(* IEC 61131-3 sources: elnaProjects/ElpcLogic/PomarKc7Changed/build_USO_ecl/_ (part 4) *)

  	IF StrSw.reliability THEN
  		IF _statOn AND NOT _statOff 		THEN 	StrSw.onStatus := _statusDualInput.STATUS_ON;
  		ELSIF _statOff AND NOT _statOn 	THEN 	StrSw.onStatus := _statusDualInput.Status_OFF;
  		ELSIF NOT _statOn AND NOT _statOff 	THEN 	StrSw.onStatus := _statusDualInput.STATUS_TRANSITIONAL;
  		ELSE					StrSw.onStatus := _statusDualInput.STATUS_ERROR;
                      END_IF;

  	ELSE
  		StrSw.onStatus := _statusDualInput.STATUS_NOTDEFINED;

  	END_IF;
  ELSE
  	CASE BYTE_TO_INT(lastCmd) OF
  		(*baseCmdOn*) 1: StrSw.onStatus  := _statusDualInput.STATUS_ON;
  		(*baseCmdOff*) 2: StrSw.onStatus  := _statusDualInput.STATUS_OFF;

  	ELSE
  		 StrSw.onStatus := _statusDualInput.STATUS_NOTDEFINED;

  	END_CASE;
  END_IF;

  StrSw.Accident := inAccident.value AND inAccident.reliability;
  StrSw.Ns := inNs.value AND inNs.reliability;
  StrSw.Local := inLocal.value AND inLocal.reliability;
  StrSw.Distance := inDistance.value AND inDistance.reliability;
  StrSw.OpcCommandsDisabled := StrSw.inOpcCommandsDisabled;

  StrSw.Blocked:=StrSw.Accident OR StrSw.Local OR StrSw.breakCmdOn OR StrSw.breakCmdOff OR StrSw.inBlocked;

  StrSw.Rezervny:=NOT StrSw.Osnovnoy;

  (* ---- Формирование признака сдвига ---- *)

  getSdvig := FALSE;
  IF (StrSw.ISVALIDREF_cmdOn OR StrSw.ISVALIDREF_cmdOff) AND NOT StrSw.Local THEN
  	IF NOT (StrSw.CmdOn OR StrSw.CmdOff) THEN
                       IF (lastOnStatus <> StrSw.onStatus AND
  		(StrSw.onStatus <> _statusDualInput.STATUS_NOTDEFINED AND
                       StrSw.onStatus <> _statusDualInput.STATUS_ERROR)     AND
  		(lastOnStatus <> _statusDualInput.STATUS_NOTDEFINED   AND
                       lastOnStatus <> _statusDualInput.STATUS_ERROR))
                      THEN
  			getSdvig   := TRUE;
  		END_IF;
  	END_IF;
  END_IF;

  IF getSdvig THEN StrSw.sdvig:= TRUE; END_IF;

  sdvigReset(IN:=StrSw.sdvig, PT:=T#15S);

  IF sdvigReset.Q THEN StrSw.sdvig:=FALSE; END_IF;

  lastOnStatus := StrSw.onStatus;

  (* ---- Распаковка команды ---- *)
  _sunpackerCommand(command := StrSw.inCommand);
  	cmd := _sunpackerCommand.cmd;
  	source := _sunpackerCommand.source;

  (* ---- Обработка команды ---- *)
  IF cmd <> 0 AND lastCmd <> cmd and (((NOT StrSw.opcCommandsDisabled) AND source > 0) OR source = 0) then
  	CASE BYTE_TO_INT(cmd) OF
  	(*cmd_on*) 1 :
  			IF  StrSw.ISVALIDREF_cmdOn THEN StrSw.CmdOn := TRUE;
  				IF StrSw.ISVALIDREF_cmdOff THEN StrSw.CmdOff := FALSE; END_IF;
  			ELSIF  StrSw.ISVALIDREF_cmdOff THEN StrSw.CmdOff := FALSE;  END_IF;
  			errorCMDTimer(IN := false);
  			_commandErrorTimer := true;
  			StrSw.lastCmdIsOn := true;
  	(*cmd_off*) 2 :
  			IF StrSw.ISVALIDREF_cmdOff THEN StrSw.CmdOff := TRUE;
  				IF StrSw.ISVALIDREF_cmdOn THEN StrSw.CmdOn := FALSE; END_IF;
  			ELSIF StrSw.ISVALIDREF_cmdOn THEN StrSw.CmdOn := FALSE; END_IF;
  			errorCMDTimer(IN := false);

  			_commandErrorTimer := true;
  			StrSw.lastCmdIsOn := false;
  	(*cmd_reset*) 3 :    IF StrSw.ISVALIDREF_statOn OR StrSw.ISVALIDREF_statOff THEN
  			StrSw.CmdOn := FALSE;
  			StrSw.CmdOff := FALSE;
                                lastCmd := 0;
  			_commandErrorTimer := false;
  			StrSw.lastCmdIsOn := false;
                                 END_IF;
  	END_CASE;
  	source_for_Status := source;
  	cmd_for_Status := cmd;
  	command_error_for_Status := 0;
  END_IF;

  lastCmd := cmd;
  errorCMDTimer(In := _commandErrorTimer, PT :=T#10s);

  (* ---- алгоритм  для команды ВКЛючить ---- *)
  IF (StrSw.onStatus = _statusDualInput.STATUS_ON) and StrSw.lastCmdIsOn then
  	IF StrSw.ISVALIDREF_cmdOn AND StrSw.ISVALIDREF_cmdOff then  StrSw.cmdOn := false; END_IF;

  	 errorCMDTimer(In := false);
  	 _commandErrorTimer := false;
  	 cmd_for_Status := 0;
  	 source_for_Status := 0;
  END_IF;

  (* ---- off ---- *)
  IF (StrSw.onStatus = _statusDualInput.STATUS_OFF) and (NOT StrSw.lastCmdIsOn) then
  	IF StrSw.ISVALIDREF_cmdOn AND StrSw.ISVALIDREF_cmdOff then  StrSw.cmdOff := false; END_IF;

  	 errorCMDTimer(In := false);
  	 _commandErrorTimer := false;
  	 cmd_for_Status := 0;
  	 source_for_Status := 0;
  END_IF;

  (* ---- ошибка исполнения команды ---- *)
  if errorCMDTimer.Q and (cmd_for_Status <> 0) then
  	command_error_for_Status :=  cmd_for_Status;
  	_commandErrorTimer := false;
  	StrSw.CmdOn := false;
  	StrSw.CmdOff := false;
  	lastCmd := 0;
  end_if;

  (* ---- сброс ошибки команды ---- *)
  StrSw.CommandFault := command_error_for_Status <> 0;
  _errorReset(IN := command_error_for_Status <> 0, PT := T#5S);
  IF _errorReset.Q THEN
  	cmd_for_Status := 0;
  	source_for_Status := 0;
  	command_error_for_Status := 0;
  END_IF;

  outputsSets(in := (StrSw.ISVALIDREF_cmdOn and StrSw.cmdOn ) OR (StrSw.ISVALIDREF_cmdOff and StrSw.cmdOff), PT := T#2S);
  	IF NOT outputsSets.Q THEN
  		StrSw.BreakCmdOn := inBreakCmdOn._inversed AND inBreakCmdOn.reliability AND StrSw.ISVALIDREF_inBreakCmdOn;
  		StrSw.BreakCmdOff := inBreakCmdOff._inversed AND inBreakCmdOff.reliability AND StrSw.ISVALIDREF_inBreakCmdOff;
  	END_IF;

  cmdOn := StrSw.cmdOn;
  cmdOff:= StrSw.cmdOff;

  (* ---- формирование зашифрованного статуса для АРМа ---- *)
  StrSw.status := shl(BYTE_TO_DWORD(source_for_Status), 29)
  		OR shl(BYTE_TO_DWORD(cmd_for_Status), 26)
  		OR shl(BYTE_TO_DWORD(command_error_for_Status), 23)
  		OR shl(bool_to_DWORD(StrSw.sdvig), 22)
  		OR shl(bool_to_DWORD(StrSw.OpcCommandsDisabled), 21)
                      OR shl(bool_to_DWORD(StrSw.lastCmdIsOn), 14)
                      OR shl(BOOL_TO_DWORD(StrSw.BreakCmdOff), 13)
  		OR shl(BOOL_TO_DWORD(StrSw.BreakCmdOn), 12)
  		OR shl(BOOL_TO_DWORD(StrSw.Distance), 6)
  		OR shl(BOOL_TO_DWORD(StrSw.Local), 5)
  		OR shl(BOOL_TO_DWORD(StrSw.Ns), 4)
                  	OR shl(BOOL_TO_DWORD(StrSw.Accident ),3)
  		OR BYTE_TO_DWORD(StrSw.onStatus);
END_FUNCTION_BLOCK

FUNCTION_BLOCK fb_Switch
  VAR_INPUT
    statOn : BOOL;
    statOff : BOOL;
    statOn_reliability : BOOL;
    statOff_reliability : BOOL;
  END_VAR
  VAR_IN_OUT
    StrSw : struct_Switch;
  END_VAR
  VAR_INPUT
    inNs : TYPE_ReliableBit;
    inAccident : TYPE_ReliableBit;
    inAuto : TYPE_ReliableBit;
    inManual : TYPE_ReliableBit;
    inLocal : TYPE_ReliableBit;
    inDistance : TYPE_ReliableBit;
    inErrorPowerOff : TYPE_ReliableBit;
    inErrorBlock : TYPE_ReliableBit;
    inBreakCmdOn : TYPE_ReliableBit;
    inBreakCmdOff : TYPE_ReliableBit;
  END_VAR
  VAR
    onInit : BOOL      := FALSE;
    _statOn : BOOL;
    _statOff : BOOL;
    lastOnStatus : BYTE;
    cmd : BYTE;
    source : BYTE;
    lastCmd : BYTE;
    source_for_Status : BYTE;
    cmd_for_Status : BYTE;
    command_error_for_Status : BYTE;
    _sunpackerCommand : fb_sunpackerCommand;
    _statusDualInput : TYPE_statusDualInput;
    _commandDualInput : TYPE_commandDualInput;
    _commandErrorTimer : BOOL;
    resetErrorTimer : BOOL;
    getSdvig : BOOL;
    _changWithoutCommand : BOOL;
    errorCMDTimer : TON;
    sdvigReset : TON;
    _errorReset : TON;
    outputsSets : TOF;
  END_VAR
  VAR_IN_OUT
    cmdOn : BOOL;
    cmdOff : BOOL;
  END_VAR

  IF NOT onInit THEN
  IF StrSw.ISVALIDREF_cmdOn XOR StrSw.ISVALIDREF_cmdOff THEN
  	IF 	StrSw.ISVALIDREF_cmdOn THEN
  		lastCmd:= 2; (*baseCmdOff*)
  	ELSE
  		lastCmd:= 1; (*baseCmdOn*)
  	END_IF;
  END_IF;
  onInit:=TRUE;
  END_IF;

  (* ---- Если управление с ВУ заблокировано, то в ИМ передаем команду из алгоритма ---- *)
  IF StrSw.inOpcCommandsDisabled THEN
  	StrSw.inCommand := StrSw.inCommand_Alg;
  ELSE (* иначе передаем команду с АРМа*)
  	StrSw.inCommand := StrSw.inCommand_ARM;
  END_IF;

  (* ---- Формирование состояния механизма ---- *)

  IF (StrSw.ISVALIDREF_statOn) OR (StrSw.ISVALIDREF_statOff) THEN
  	IF (StrSw.ISVALIDREF_statOn) AND (StrSw.ISVALIDREF_statOff) THEN
  	StrSw.reliability:= statOn_reliability AND statOff_reliability;
  		_statOn  := statOn;
  		_statOff := statOff;
  	ELSIF (StrSw.ISVALIDREF_statOn) THEN
                       StrSw.reliability:= statOn_reliability;
  		_statOn  := statOn;
  		_statOff := NOT statOn;
  	ELSIF (StrSw.ISVALIDREF_statOff) THEN
  		 StrSw.reliability:= statOff_reliability;
  		_statOn  := NOT statOff;
  		_statOff :=statOff;
  	END_IF;

  	IF StrSw.reliability THEN
  		IF _statOn AND NOT _statOff 		THEN 	StrSw.onStatus := _statusDualInput.STATUS_ON;
  		ELSIF _statOff AND NOT _statOn 	THEN 	StrSw.onStatus := _statusDualInput.Status_OFF;
  		ELSIF NOT _statOn AND NOT _statOff 	THEN 	StrSw.onStatus := _statusDualInput.STATUS_TRANSITIONAL;
  		ELSE					StrSw.onStatus := _statusDualInput.STATUS_ERROR;
                      END_IF;

  	ELSE
  		StrSw.onStatus := _statusDualInput.STATUS_NOTDEFINED;

  	END_IF;
  ELSE
  	CASE BYTE_TO_INT(lastCmd) OF
  		(*baseCmdOn*) 1: StrSw.onStatus  := _statusDualInput.STATUS_ON;
  		(*baseCmdOff*) 2: StrSw.onStatus  := _statusDualInput.STATUS_OFF;

  	ELSE
  		 StrSw.onStatus := _statusDualInput.STATUS_NOTDEFINED;

  	END_CASE;
  END_IF;

  StrSw.Accident := inAccident.value AND inAccident.reliability;
  StrSw.Ns := inNs.value AND inNs.reliability;
  StrSw.Auto := inAuto.value AND inAuto.reliability;
  StrSw.Manual := inManual.value AND inManual.reliability;
  StrSw.Local := inLocal.value AND inLocal.reliability;
  StrSw.Distance := inDistance.value AND inDistance.reliability;
  StrSw.ErrorPowerOff := inErrorPowerOff.value AND inErrorPowerOff.reliability;
  StrSw.ErrorBlock := inErrorBlock.value AND inErrorBlock.reliability;
  StrSw.OpcCommandsDisabled := StrSw.inOpcCommandsDisabled;

  (* ---- Формирование признака сдвига ---- *)
  getSdvig := FALSE;
  IF (StrSw.ISVALIDREF_cmdOn OR StrSw.ISVALIDREF_cmdOff) AND NOT StrSw.Local THEN
  	IF NOT (StrSw.CmdOn OR StrSw.CmdOff) THEN
                       IF (lastOnStatus <> StrSw.onStatus AND
  		(StrSw.onStatus <> _statusDualInput.STATUS_NOTDEFINED AND
                       StrSw.onStatus <> _statusDualInput.STATUS_ERROR)     AND
  		(lastOnStatus <> _statusDualInput.STATUS_NOTDEFINED   AND
                       lastOnStatus <> _statusDualInput.STATUS_ERROR))
                      THEN
  			getSdvig   := TRUE;
  		END_IF;
  	END_IF;
  END_IF;

  IF getSdvig THEN StrSw.sdvig:= TRUE; END_IF;

  sdvigReset(IN:=StrSw.sdvig, PT:=T#15S);

  IF sdvigReset.Q THEN StrSw.sdvig:=FALSE; END_IF;

  lastOnStatus := StrSw.onStatus;

  (* ---- Распаковка команды ---- *)
  _sunpackerCommand(command := StrSw.inCommand);
  	cmd := _sunpackerCommand.cmd;
  	source := _sunpackerCommand.source;

  (* ---- Обработка команды ---- *)
  IF cmd <> 0 AND lastCmd <> cmd and (((NOT StrSw.opcCommandsDisabled) AND source > 0) OR source = 0) then
  	CASE BYTE_TO_INT(cmd) OF
  	(*cmd_open*) 1 :
  			IF  StrSw.ISVALIDREF_cmdOn THEN StrSw.CmdOn := TRUE;
  				IF StrSw.ISVALIDREF_cmdOff THEN StrSw.CmdOff := FALSE; END_IF;
  			ELSIF  StrSw.ISVALIDREF_cmdOff THEN StrSw.CmdOff := FALSE;  END_IF;
                                lastCmd := cmd;
  			errorCMDTimer(IN := false);
  			_commandErrorTimer := true;
  			StrSw.lastCmdIsOn := true;
  	(*cmd_close*) 2 :
  			IF StrSw.ISVALIDREF_cmdOff THEN StrSw.CmdOff := TRUE;
  				IF StrSw.ISVALIDREF_cmdOn THEN StrSw.CmdOn := FALSE; END_IF;
  			ELSIF StrSw.ISVALIDREF_cmdOn THEN StrSw.CmdOn := FALSE; END_IF;
                                lastCmd := cmd;
  			errorCMDTimer(IN := false);
  			_commandErrorTimer := true;
  			StrSw.lastCmdIsOn := false;
  	(*cmd_reset*) 3 :    IF StrSw.ISVALIDREF_statOn OR StrSw.ISVALIDREF_statOff THEN
  			StrSw.CmdOn := FALSE;
  			StrSw.CmdOff := FALSE;
                                lastCmd :=0;
  			_commandErrorTimer := false;
  			StrSw.lastCmdIsOn := false;
                                 END_IF;
  	END_CASE;
  	source_for_Status := source;
  	cmd_for_Status := cmd;
  	command_error_for_Status := 0;
  END_IF;

  errorCMDTimer(In := _commandErrorTimer, PT :=T#10s);

  (* ---- алгоритм  для команды ВКЛючить ---- *)
  IF (StrSw.onStatus = _statusDualInput.STATUS_ON) and StrSw.lastCmdIsOn then
  	IF StrSw.ISVALIDREF_cmdOn AND StrSw.ISVALIDREF_cmdOff then  StrSw.cmdOn := false; END_IF;

  	 errorCMDTimer(In := false);
  	 _commandErrorTimer := false;
  	 cmd_for_Status := 0;
  	 source_for_Status := 0;
  END_IF;

  (* ---- off ---- *)
  IF (StrSw.onStatus = _statusDualInput.STATUS_OFF) and (NOT StrSw.lastCmdIsOn) then
  	IF StrSw.ISVALIDREF_cmdOn AND StrSw.ISVALIDREF_cmdOff then  StrSw.cmdOff := false; END_IF;

  	 errorCMDTimer(In := false);
  	 _commandErrorTimer := false;
  	 cmd_for_Status := 0;
  	 source_for_Status := 0;
  END_IF;

  (* ---- ошибка исполнения команды ---- *)
  if errorCMDTimer.Q and (cmd_for_Status <> 0) then
  	command_error_for_Status :=  cmd_for_Status;
  	_commandErrorTimer := false;
  	StrSw.CmdOn := false;
  	StrSw.CmdOff := false;
  	lastCmd := 0;
  end_if;

  (* ---- сброс ошибки команды ---- *)
  StrSw.CommandFault := command_error_for_Status <> 0;
  _errorReset(IN := command_error_for_Status <> 0, PT := T#5S);
  IF _errorReset.Q THEN
  	cmd_for_Status := 0;
  	source_for_Status := 0;
  	command_error_for_Status := 0;
  END_IF;

  outputsSets(in := (StrSw.ISVALIDREF_cmdOn and StrSw.cmdOn ) OR (StrSw.ISVALIDREF_cmdOff and StrSw.cmdOff), PT := T#2S);
  	IF NOT outputsSets.Q THEN
  		StrSw.BreakCmdOn := inBreakCmdOn._inversed AND
                      inBreakCmdOn.reliability AND StrSw.ISVALIDREF_inBreakCmdOn;

  		StrSw.BreakCmdOff := inBreakCmdOff._inversed
                      AND inBreakCmdOff.reliability AND StrSw.ISVALIDREF_inBreakCmdOff;
  	END_IF;

  cmdOn := StrSw.cmdOn;
  cmdOff:= StrSw.cmdOff;

  (* ---- формирование зашифрованного статуса для АРМа ---- *)
  StrSw.status := shl(BYTE_TO_DWORD(source_for_Status), 29)
  		OR shl(BYTE_TO_DWORD(cmd_for_Status), 26)
  		OR shl(BYTE_TO_DWORD(command_error_for_Status), 23)
  		OR shl(bool_to_DWORD(StrSw.sdvig), 22)
  		OR shl(bool_to_DWORD(StrSw.OpcCommandsDisabled), 21)
                      OR shl(bool_to_DWORD(StrSw.lastCmdIsOn), 14)
                      OR shl(BOOL_TO_DWORD(StrSw.BreakCmdOff), 13)
  		OR shl(BOOL_TO_DWORD(StrSw.BreakCmdOn), 12)
  		OR shl(BOOL_TO_DWORD(StrSw.ErrorBlock), 11)
  		OR shl(BOOL_TO_DWORD(StrSw.ErrorPowerOff), 10)
  		OR shl(BOOL_TO_DWORD(StrSw.Manual), 8)
  		OR shl(BOOL_TO_DWORD(StrSw.Auto), 7)
  		OR shl(BOOL_TO_DWORD(StrSw.Distance), 6)
  		OR shl(BOOL_TO_DWORD(StrSw.Local), 5)
  		OR shl(BOOL_TO_DWORD(StrSw.Ns), 4)
                  	OR shl(BOOL_TO_DWORD(StrSw.Accident ),3)
  		OR BYTE_TO_DWORD(StrSw.onStatus);
END_FUNCTION_BLOCK

FUNCTION_BLOCK fb_SectionSwitch
  VAR_INPUT
    statOn : BOOL;
    statOff : BOOL;
    statOn_reliability : BOOL;
    statOff_reliability : BOOL;
  END_VAR
  VAR_IN_OUT
    StrSw : struct_SectionSwitch;
  END_VAR
  VAR_INPUT
    basketRolledIn : TYPE_ReliableBit;
    basketRolledOut : TYPE_ReliableBit;
    basketTest : TYPE_ReliableBit;
    inNs : TYPE_ReliableBit;
    inoffKNA : TYPE_ReliableBit;
    inAccident : TYPE_ReliableBit;
    inLocal : TYPE_ReliableBit;
    inDistance : TYPE_ReliableBit;
    inBreakCmdOn : TYPE_ReliableBit;
    inBreakCmdOff : TYPE_ReliableBit;
  END_VAR
  VAR
    onInit : BOOL      := FALSE;
    _statOn : BOOL;
    _statOff : BOOL;
    getSdvig : BOOL;
    lastOnStatus : BYTE;
    cmd : BYTE;
    source : BYTE;
    lastCmd : BYTE;
    source_for_Status : BYTE;
    cmd_for_Status : BYTE;
    command_error_for_Status : BYTE;
    _basketRolledIn : TYPE_ReliableBit;
    _basketRolledOut : TYPE_ReliableBit;
    _basketTest : TYPE_ReliableBit;
    _sunpackerCommand : fb_sunpackerCommand;
    _statusDualInput : TYPE_statusDualInput;
    _statusBasket : TYPE_basketStats;
    _commandDualInput : TYPE_commandDualInput;
    _commandErrorTimer : BOOL;
    resetErrorTimer : BOOL;
    _changWithoutCommand : BOOL;
    errorCMDTimer : TON;
    _errorReset : TON;
    sdvigReset : TON;
    outputsSets : TOF;
  END_VAR
  VAR_IN_OUT
    cmdOn : BOOL;
    cmdOff : BOOL;
  END_VAR

  IF NOT onInit THEN
  IF StrSw.ISVALIDREF_cmdOn XOR StrSw.ISVALIDREF_cmdOff THEN
  	IF 	StrSw.ISVALIDREF_cmdOn THEN
  		lastCmd:= 2; (*baseCmdOff*)
  	ELSE
  		lastCmd:= 1; (*baseCmdOn*)
  	END_IF;
  END_IF;
  onInit:=TRUE;
  END_IF;

  (* ---- Формирование состояния тележки ---- *)

  IF (NOT StrSw.ISVALIDREF_basketRolledIn) AND (NOT StrSw.ISVALIDREF_basketRolledOut) THEN
            StrSw.basketStatus:=_statusBasket.BASKET_NOTDEFINED;
  ELSE
  		IF StrSw.ISVALIDREF_basketTest THEN
  		_basketTest:=basketTest;
  	ELSE
  		_basketTest.reliability:=TRUE;
  		_basketTest.value :=FALSE;
  	END_IF;

  	IF StrSw.ISVALIDREF_basketRolledIn THEN
  		_basketRolledIn:=basketRolledIn;
  	ELSE
  		_basketRolledIn:=basketRolledOut;
  		IF StrSw.ISVALIDREF_basketTest THEN
  		_basketRolledIn.value:=NOT (_basketRolledIn.value OR _basketTest.value);
  		ELSE
  		_basketRolledIn.value:= NOT _basketRolledIn.value;
  		END_IF;

  	END_IF;

  	IF StrSw.ISVALIDREF_basketRolledOut THEN
  		_basketRolledOut:=basketRolledOut;
  	ELSE
  		_basketRolledOut:=basketRolledIn;
  		IF StrSw.ISVALIDREF_basketTest THEN
  		_basketRolledOut.value:= NOT (_basketRolledOut.value OR _basketTest.value );
  		ELSE
  			_basketRolledOut.value := NOT _basketRolledout.value;
  		END_IF;

  	END_IF;

  IF _basketRolledIn.reliability AND _basketRolledOut.reliability AND _basketTest.reliability THEN
  		IF (BOOL_TO_INT(_basketRolledIn.value)+BOOL_TO_INT(_basketRolledOut.value)+BOOL_TO_INT(_basketTest.value))=1 THEN
  			IF _basketRolledIn.value THEN
  				StrSw.basketStatus:=_statusBasket.BASKET_ROLLEDIN;
  			ELSIF _basketRolledOut.value THEN
  				StrSw.basketStatus:=_statusBasket.BASKET_ROLLEDOUT;
  			ELSIF _basketTest.value THEN
  				StrSw.basketStatus:=_statusBasket.BASKET_TEST;
  			END_IF;
  		ELSE
  			StrSw.basketStatus:=_statusBasket.BASKET_ERROR;
  		END_IF;
  	ELSE
  		StrSw.basketStatus:=_statusBasket.BASKET_NOTDEFINED;
  	END_IF;
  END_IF;

  (* ---- Если управление с ВУ заблокировано, то в ИМ передаем команду из алгоритма ---- *)
  IF StrSw.inOpcCommandsDisabled THEN
  	StrSw.inCommand := StrSw.inCommand_Alg;
  ELSE (* иначе передаем команду с АРМа*)
  	StrSw.inCommand := StrSw.inCommand_ARM;
  END_IF;

  (* ---- Формирование состояния механизма ---- *)

  IF (StrSw.ISVALIDREF_statOn) OR (StrSw.ISVALIDREF_statOff) THEN
  	IF (StrSw.ISVALIDREF_statOn) AND (StrSw.ISVALIDREF_statOff) THEN
  	StrSw.reliability:= statOn_reliability AND statOff_reliability;
  		_statOn  := statOn;
  		_statOff := statOff;
  	ELSIF (StrSw.ISVALIDREF_statOn) THEN
                       StrSw.reliability:= statOn_reliability;
  		_statOn  := statOn;
  		_statOff := NOT statOn;
  	ELSIF (StrSw.ISVALIDREF_statOff) THEN
  		 StrSw.reliability:= statOff_reliability;
  		_statOn  := NOT statOff;
  		_statOff :=statOff;
  	END_IF;

  	IF StrSw.reliability THEN
  		IF _statOn AND NOT _statOff 		THEN 	StrSw.onStatus := _statusDualInput.STATUS_ON;
  		ELSIF _statOff AND NOT _statOn 	THEN 	StrSw.onStatus := _statusDualInput.Status_OFF;
  		ELSIF NOT _statOn AND NOT _statOff 	THEN 	StrSw.onStatus := _statusDualInput.STATUS_TRANSITIONAL;
  		ELSE					StrSw.onStatus := _statusDualInput.STATUS_ERROR;
                      END_IF;

  	ELSE
  		StrSw.onStatus := _statusDualInput.STATUS_NOTDEFINED;

  	END_IF;
  ELSE
  	CASE BYTE_TO_INT(lastCmd) OF
  		(*baseCmdOn*) 1: StrSw.onStatus  := _statusDualInput.STATUS_ON;
  		(*baseCmdOff*) 2: StrSw.onStatus  := _statusDualInput.STATUS_OFF;

  	ELSE
  		 StrSw.onStatus := _statusDualInput.STATUS_NOTDEFINED;

  	END_CASE;
  END_IF;

  StrSw.Accident := inAccident.value AND inAccident.reliability;
  StrSw.Ns := inNs.value AND inNs.reliability;
  StrSw.Local := inLocal.value AND inLocal.reliability;
  StrSw.Distance := inDistance.value AND inDistance.reliability;
  StrSw.OpcCommandsDisabled := StrSw.inOpcCommandsDisabled;
  StrSw.offKNA := inoffKNA.value AND inoffKNA.reliability;

  (* ---- Формирование признака сдвига ---- *)

  getSdvig := FALSE;
  IF (StrSw.ISVALIDREF_cmdOn OR StrSw.ISVALIDREF_cmdOff) AND NOT StrSw.Local THEN
  	IF NOT (StrSw.CmdOn OR StrSw.CmdOff) THEN
                       IF (lastOnStatus <> StrSw.onStatus AND
  		(StrSw.onStatus <> _statusDualInput.STATUS_NOTDEFINED AND
                       StrSw.onStatus <> _statusDualInput.STATUS_ERROR)     AND
  		(lastOnStatus <> _statusDualInput.STATUS_NOTDEFINED   AND
                       lastOnStatus <> _statusDualInput.STATUS_ERROR))
                      THEN
  			getSdvig   := TRUE;
  		END_IF;
  	END_IF;
  END_IF;

  IF getSdvig THEN StrSw.sdvig:= TRUE; END_IF;

  sdvigReset(IN:=StrSw.sdvig, PT:=T#15S);

  IF sdvigReset.Q THEN StrSw.sdvig:=FALSE; END_IF;

  lastOnStatus := StrSw.onStatus;

  (* ---- Распаковка команды ---- *)
  _sunpackerCommand(command := StrSw.inCommand);
  	cmd := _sunpackerCommand.cmd;
  	source := _sunpackerCommand.source;

  (* ---- Обработка команды ---- *)
  IF cmd <> 0 AND lastCmd <> cmd and (((NOT StrSw.opcCommandsDisabled) AND source > 0) OR source = 0) then
  	CASE BYTE_TO_INT(cmd) OF
  	(*cmd_open*) 1 :
  			IF  StrSw.ISVALIDREF_cmdOn THEN StrSw.CmdOn := TRUE;
  				IF StrSw.ISVALIDREF_cmdOff THEN StrSw.CmdOff := FALSE; END_IF;
  			ELSIF  StrSw.ISVALIDREF_cmdOff THEN StrSw.CmdOff := FALSE;  END_IF;
  			errorCMDTimer(IN := false);
  			_commandErrorTimer := true;
  			StrSw.lastCmdIsOn := true;
  	(*cmd_close*) 2 :
  			IF StrSw.ISVALIDREF_cmdOff THEN StrSw.CmdOff := TRUE;
  				IF StrSw.ISVALIDREF_cmdOn THEN StrSw.CmdOn := FALSE; END_IF;
  			ELSIF StrSw.ISVALIDREF_cmdOn THEN StrSw.CmdOn := FALSE; END_IF;
  			errorCMDTimer(IN := false);
  			_commandErrorTimer := true;
  			StrSw.lastCmdIsOn := false;
  	(*cmd_reset*) 3 :    IF StrSw.ISVALIDREF_statOn OR StrSw.ISVALIDREF_statOff THEN
  			StrSw.CmdOn := FALSE;
  			StrSw.CmdOff := FALSE;
                                lastCmd := 0;
  			_commandErrorTimer := false;
  			StrSw.lastCmdIsOn := false;
                                 END_IF;
  	END_CASE;
  	source_for_Status := source;
  	cmd_for_Status := cmd;
  	command_error_for_Status := 0;
  END_IF;
  lastCmd := cmd;

  errorCMDTimer(In := _commandErrorTimer, PT :=T#10s);

  (* ---- алгоритм  для команды ВКЛючить ---- *)
  IF (StrSw.onStatus = _statusDualInput.STATUS_ON) and (StrSw.lastCmdIsOn) then
  	IF StrSw.ISVALIDREF_cmdOn AND StrSw.ISVALIDREF_cmdOff then  StrSw.cmdOn := false; END_IF;

  	 errorCMDTimer(In := false);
  	 _commandErrorTimer := false;
  	 cmd_for_Status := 0;
  	 source_for_Status := 0;
  END_IF;

  (* ---- off ---- *)
  IF (StrSw.onStatus = _statusDualInput.STATUS_OFF) and (NOT StrSw.lastCmdIsOn) then
  	IF StrSw.ISVALIDREF_cmdOn AND StrSw.ISVALIDREF_cmdOff then  StrSw.cmdOff := false; END_IF;

  	 errorCMDTimer(In := false);
  	 _commandErrorTimer := false;
  	 cmd_for_Status := 0;
  	 source_for_Status := 0;
  END_IF;

  (* ---- ошибка исполнения команды ---- *)
  if errorCMDTimer.Q and (cmd_for_Status <> 0) then
  	command_error_for_Status :=  cmd_for_Status;
  	_commandErrorTimer := false;
  	StrSw.CmdOn := false;
  	StrSw.CmdOff := false;
  	lastCmd := 0;
  end_if;

  (* ---- сброс ошибки команды ---- *)
  StrSw.CommandFault := command_error_for_Status <> 0;
  _errorReset(IN := command_error_for_Status <> 0, PT := T#5S);
  IF _errorReset.Q THEN
  	cmd_for_Status := 0;
  	source_for_Status := 0;
  	command_error_for_Status := 0;
  END_IF;

  outputsSets(in := (StrSw.ISVALIDREF_cmdOn and StrSw.cmdOn ) OR (StrSw.ISVALIDREF_cmdOff and StrSw.cmdOff), PT := T#2S);
  	IF NOT outputsSets.Q THEN
  		StrSw.BreakCmdOn := inBreakCmdOn._inversed AND inBreakCmdOn.reliability AND StrSw.ISVALIDREF_inBreakCmdOn;
  		StrSw.BreakCmdOff := inBreakCmdOff._inversed AND inBreakCmdOff.reliability AND StrSw.ISVALIDREF_inBreakCmdOff;
  	END_IF;

  cmdOn := StrSw.cmdOn;
  cmdOff:= StrSw.cmdOff;

  (* ---- формирование зашифрованного статуса для АРМа ---- *)
  StrSw.status := shl(BYTE_TO_DWORD(source_for_Status), 29)
  		OR shl(BYTE_TO_DWORD(cmd_for_Status), 26)
  		OR shl(BYTE_TO_DWORD(command_error_for_Status), 23)
  		OR shl(bool_to_DWORD(StrSw.sdvig), 22)
  		OR shl(bool_to_DWORD(StrSw.OpcCommandsDisabled), 21)
                      OR shl(BOOL_TO_DWORD(StrSw.offKNA), 17)
                      OR shl(bool_to_DWORD(StrSw.lastCmdIsOn), 14)
                      OR shl(BOOL_TO_DWORD(StrSw.BreakCmdOff), 13)
  		OR shl(BOOL_TO_DWORD(StrSw.BreakCmdOn), 12)
                      OR shl(BYTE_TO_DWORD(StrSw.basketStatus), 8)
  		OR shl(BOOL_TO_DWORD(StrSw.Distance), 6)
  		OR shl(BOOL_TO_DWORD(StrSw.Local), 5)
  		OR shl(BOOL_TO_DWORD(StrSw.Ns), 4)
                  	OR shl(BOOL_TO_DWORD(StrSw.Accident ),3)
  		OR BYTE_TO_DWORD(StrSw.onStatus);
END_FUNCTION_BLOCK

FUNCTION_BLOCK fb_singleSignal
  VAR_INPUT
    signal : TYPE_ReliableBit;
  END_VAR
  VAR_IN_OUT
    str_SS : struct_singleSignal;
  END_VAR
  VAR
    TimerOn : TON;
    TimerOff : TOF;
  END_VAR

  str_SS.reliability:=signal.reliability;

  IF NOT str_SS.inverse THEN
  TimerOn(IN:=(signal.value AND str_SS.reliability AND NOT str_SS.Disabled_Sig), PT:=str_SS.DelayOn);
  ELSE
  TimerOn(IN:=(signal._inversed AND str_SS.reliability AND NOT str_SS.Disabled_Sig), PT:=str_SS.DelayOn);
  END_IF;

  TimerOff(IN:=TimerOn.Q, PT:=str_SS.DelayOff);

  str_SS.Q:=TimerOff.Q;

  str_SS.status:= SHL(BOOL_TO_DWORD(NOT str_SS.reliability), 15)
  	OR BOOL_TO_DWORD(str_SS.Q);
END_FUNCTION_BLOCK

FUNCTION_BLOCK fb_singleOutput
  VAR_IN_OUT
    signal : BOOL;
    str_SO : struct_singleOutput;
  END_VAR
  VAR
    pulseTimer : TON;
    resetCmdTimer : TON;
    TON_Command : TON;
    source : BYTE;
    cmd : BYTE;
    lastCmd : BYTE;
    source_for_Status : BYTE;
    cmd_for_Status : BYTE;
    command_error_for_Status : BYTE;
    pulseTimerPriznak : BOOL;
    resetCmdTimerPriznak : BOOL;
    _sunpackerCommand : fb_sunpackerCommand;
  END_VAR

  str_SO.OpcCommandsDisabled := str_SO.inOpcCommandsDisabled;

  (* ---- Если управление с ВУ заблокировано, то передаем команду из алгоритма ---- *)
  IF str_SO.inOpcCommandsDisabled THEN
  	str_SO.inCommand := str_SO.inCommand_Alg;
  ELSE (* иначе передаем команду с АРМа*)
  	str_SO.inCommand := str_SO.inCommand_ARM;
  END_IF;

  (*Распаковка команды*)
  _sunpackerCommand(command := str_SO.inCommand);
  	cmd := _sunpackerCommand.cmd;
  	source := _sunpackerCommand.source;

  (*Обработка команды*)
  IF cmd <> 0 AND lastCmd <> cmd and (((NOT str_SO.OpcCommandsDisabled) AND source > 0) OR source = 0) then
  	CASE BYTE_TO_INT(cmd) OF
  	(*cmd_on*) 1 :
  			str_SO.Q := TRUE;
  			pulseTimer(IN := FALSE);
  			pulseTimerPriznak := FALSE;
  			resetCmdTimer(IN := FALSE);
  			resetCmdTimerPriznak := TRUE;
  	(*cmd_off*) 2 :
  			str_SO.Q := FALSE;
  			pulseTimer(IN := FALSE);
  			pulseTimerPriznak := FALSE;
  			resetCmdTimer(IN := FALSE);
  			resetCmdTimerPriznak := TRUE;
  	(*cmd_pulse*) 3 :
  			str_SO.Q := TRUE;
                                pulseTimer(IN := FALSE);
                                pulseTimerPriznak := TRUE;
  			resetCmdTimer(IN := FALSE);
                                resetCmdTimerPriznak := FALSE;
  	END_CASE;
  	source_for_Status := source;
  	cmd_for_Status := cmd;
  	command_error_for_Status := 0;
  END_IF;
  lastCmd := cmd;

  pulseTimer(IN := pulseTimerPriznak, PT := str_SO.wait_time);
  pulseTimer();
  IF pulseTimer.Q THEN
  	pulseTimer(IN := FALSE);
  	pulseTimerPriznak := FALSE;

  	str_SO.Q := FALSE;

  	source_for_Status := 0;
  	cmd_for_Status := 0;
  	command_error_for_Status := 0;
  END_IF;

  resetCmdTimer(IN := resetCmdTimerPriznak, PT := T#10S);
  resetCmdTimer();
  IF resetCmdTimer.Q THEN
  	resetCmdTimer(IN := FALSE);
  	resetCmdTimerPriznak := FALSE;

  	source_for_Status := 0;
  	cmd_for_Status := 0;
  	command_error_for_Status := 0;
  END_IF;

  signal:= str_SO.Q;

  (*TON_Command(IN:= (inCommand <> 0) AND (source = 0), PT:= T#2S);*)
      (*IF TON_Command.Q THEN*)
          (*inCommand := 0;*)
      (*END_IF;*)
  str_SO.status :=                           shl(BYTE_TO_DWORD(source_for_Status), 29)
  				OR shl(BYTE_TO_DWORD(cmd_for_Status), 26)
  				OR shl(BYTE_TO_DWORD(command_error_for_Status), 23)
  				OR shl(BOOL_TO_DWORD(str_SO.OpcCommandsDisabled), 21)
  				OR BOOL_TO_DWORD(str_SO.Q);
END_FUNCTION_BLOCK

FUNCTION_BLOCK proc_IM
  VAR
    fb_Kran1 : fb_Kran;
    fb_Kran2 : fb_Kran;
    fb_Kran3 : fb_Kran;
    fb_Kran3b : fb_Kran;
    fb_Kran4 : fb_Kran;
    fb_Kran5 : fb_Kran;
    fb_Kran6 : fb_Kran;
    fb_nu1 : fb_OilPump;
    fb_nu2 : fb_OilPump;
    fb_pns : fb_Switch;
    fb_v1_Avom : fb_Switch;
    fb_v2_Avom : fb_Switch;
    fb_v3_Avom : fb_Switch;
    fb_v4_Avom : fb_Switch;
    fb_TEN_kollectora : fb_Switch;
    fb_KaloriferAVOM : fb_Switch;
    fb_CMN : fb_Switch;
    fb_TEN_MB : fb_Switch;
    fb_mv : fb_SectionSwitch;
    fb_PLC_Control : fb_meandr;
  END_VAR
  VAR_EXTERNAL
    di : DiConfig;
    od : DOconfig;
    IM : ImConfig;
  END_VAR
  VAR
    fb_dP_maslo_gaz_Less100 : fb_singleSignal;
    fb_dp_kran1_Less100 : fb_singleSignal;
    fb_QF1_on : fb_singleSignal;
    fb_QF2_on : fb_singleSignal;
    fb_QF23_on : fb_singleSignal;
    fb_QF4_QF5_on : fb_singleSignal;
    fb_QF6_QF7_on : fb_singleSignal;
    fb_QF8_QF9_on : fb_singleSignal;
    fb_QF10_QF11_on : fb_singleSignal;
    fb_QF12_QF13_on : fb_singleSignal;
    fb_QF14_QF15_on : fb_singleSignal;
    fb_QF22_on : fb_singleSignal;
    fb_NS_G1_G2 : fb_singleSignal;
    fb_NS_G3_G4 : fb_singleSignal;
    fb_NS_G15_G16 : fb_singleSignal;
    fb_NS_G17 : fb_singleSignal;
    fb_NS_G5_G6 : fb_singleSignal;
    fb_NS_G7_G8 : fb_singleSignal;
    fb_NS_G18_G19 : fb_singleSignal;
    fb_NS_G10_G11 : fb_singleSignal;
    fb_NS_G13_G14 : fb_singleSignal;
    fb_Vozbud_neispr_tsepey_upr_AVR_pit : fb_singleSignal;
    fb_Vozbud_gotovnost : fb_singleSignal;
    fb_Vozbud_neispravnost : fb_singleSignal;
    fb_SHAVR1_v_rabote : fb_singleSignal;
    fb_SHAVR2_v_rabote : fb_singleSignal;
    fb_Avariinoe_otkluch_vikluchatelya : fb_singleSignal;
    fb_Assinhronnii_hod_peregruzka : fb_singleSignal;
    fb_SHU_v_GPA_vkluch : fb_singleSignal;
    fb_SHP_v_GPA_vkluch : fb_singleSignal;
    fb_Uroven_masla_akkum : fb_singleSignal;
    fb_NKU1_GPA_on : fb_singleSignal;
    fb_NKU2_GPA_on : fb_singleSignal;
    fb_AO_KC_ot_SHKS : fb_singleSignal;
    fb_AO_GPA_ot_SHU : fb_singleSignal;
    fb_BEAO_srabotal : fb_singleSignal;
    fb_Chastotny_pusk : fb_singleSignal;
    fb_Neuspesh_chastotny_pusk : fb_singleSignal;
    fb_Rezhim_ruchnogo_regulirovaniya : fb_singleSignal;
    fb_Razreshenie_zagruzki_dvig : fb_singleSignal;
    fb_Osnovnoy_regul_off : fb_singleSignal;
    fb_Voltage_sekcii_norm : fb_singleSignal;
    fb_Reactorny_pusk : fb_singleSignal;
    fb_NO_GPA_ot_SHU : fb_singleSignal;
    fb_AO_GPA_ot_PRU : fb_singleSignal;
    fb_Nalichie_BP1 : fb_singleSignal;
    fb_Nalichie_BP2 : fb_singleSignal;
    fb_Nalichie_BP3 : fb_singleSignal;
    fb_Nalichie_BP4 : fb_singleSignal;
    fb_Nalichie_BP5 : fb_singleSignal;
    fb_Nalichie_BP6 : fb_singleSignal;
    fb_Nalichie_BP7_BP8 : fb_singleSignal;
    fb_Nalichie_BP9_BP10 : fb_singleSignal;
    fb_Nalichie_cepei_upravlen_mv : fb_singleSignal;
    fb_Nalichie_220BEAO : fb_singleSignal;
    fb_Nalichie_per_220_na_vhode : fb_singleSignal;
    fb_Nalichie_post_220_na_vhode : fb_singleSignal;
    fb_Nalichie_BP11 : fb_singleSignal;
    fb_Nalichie_BP12 : fb_singleSignal;
    fb_Dver_SHU_pered_otkrita : fb_singleSignal;
    fb_Dver_SHU_zad_otkrita : fb_singleSignal;
    fb_EO_GPA_ot_knopki_SHU : fb_singleSignal;
    fb_EO_EGPA_ot_PRY : fb_singleSignal;
    fb_Synchroniz_rezhima_K1 : fb_singleSignal;
    fb_Potok_ms_posle_AVOM : fb_singleSignal;
    fb_Avary_EGPA : fb_singleOutput;
    fb_U_lamp_SHU : fb_singleOutput;
    fb_AO_knopka_ind : fb_singleOutput;
    fb_Pusk : fb_singleOutput;
    fb_Stop_SHUP : fb_singleOutput;
    fb_NO_fonar : fb_singleOutput;
    fb_PC_fonar : fb_singleOutput;
    fb_AC_fonar : fb_singleOutput;
    fb_Kr1_smazka : fb_singleOutput;
    fb_Kr2_smazka : fb_singleOutput;
    fb_Kr4_open_from_alg : fb_singleOutput;
    fb_Synch_rej_K1 : fb_singleOutput;
    fb_Rabota_EGPA : fb_singleOutput;
    fb_Neispr_EGPA : fb_singleOutput;
  END_VAR

  (* Циклический опрос. ИМ *)

  (* GPIO *)
  fb_PLC_Control(output:=od.gpio_out.bits[0]);

  (* Кран 1 *)
  fb_Kran1(statOn := di.di_20.bits[5]._inversed,
           statOff := di.di_20.bits[4]._inversed,
           inSo := di.di_16.bits[0], inSz := di.di_16.bits[1],
           cmdOn:=od.do_0.bits[0], cmdOff:=od.do_0.bits[1],
           strKr:= IM.Kran1  );

  (* Кран 2 *)
  fb_Kran2(statOn := di.di_21.bits[0]._inversed,
           statOff := di.di_20.bits[7]._inversed,
           inSo := di.di_16.bits[2], inSz := di.di_16.bits[3],
           cmdOn:=od.do_0.bits[2], cmdOff:=od.do_0.bits[3],
           strKr:= IM.Kran2  );

  (* Кран 3 *)
  fb_Kran3(statOn := di.di_0.bits[5]._inversed,
           statOff := di.di_0.bits[4]._inversed,
           inSo := di.di_16.bits[4], inSz := di.di_16.bits[5],
           cmdOn:=od.do_0.bits[4], cmdOff:=od.do_0.bits[5],
           strKr:= IM.Kran3  );

  (* Кран 3b *)
  fb_Kran3b(statOn := di.di_0.bits[7]._inversed,
           statOff := di.di_0.bits[6]._inversed,
           inSo := di.di_16.bits[6], inSz := di.di_16.bits[7],
           cmdOn:=od.do_0.bits[6], cmdOff:=od.do_0.bits[7],
           strKr:= IM.Kran3b  );

  (* Кран 4 *)
  fb_Kran4(statOn := di.di_1.bits[1]._inversed,
           statOff := di.di_1.bits[0]._inversed,
           inSo := di.di_17.bits[0], inSz := di.di_17.bits[1],
           cmdOn:=od.do_0.bits[8], cmdOff:=od.do_0.bits[9],
           strKr:= IM.Kran4  );

  (* Кран 5 *)
  fb_Kran5(statOn := di.di_1.bits[3]._inversed,
           statOff := di.di_1.bits[2]._inversed,
           inSo := di.di_17.bits[2], inSz := di.di_17.bits[3],
           cmdOn:=od.do_0.bits[10], cmdOff:=od.do_0.bits[11],
           strKr:= IM.Kran5  );

  (* Кран 6НР *)
  fb_Kran6(statOn := di.di_1.bits[5]._inversed,
           statOff := di.di_1.bits[4]._inversed,
           inSo := di.di_17.bits[4], inSz := di.di_17.bits[5],
           cmdOn:=od.do_0.bits[12], cmdOff:=od.do_0.bits[13],
           strKr:= IM.Kran6  );

  (*  НУ1 Насос уплотнения *)
  fb_nu1(statOn := di.di_5.bits[1].value, statOff := di.di_5.bits[1]._inversed,
           cmdOn:=od.do_1.bits[4], cmdOff:=od.do_1.bits[5],
           StrSw:= IM.nu1  );

  (*  НУ2 Насос уплотнения *)
  fb_nu2(statOn := di.di_5.bits[2].value, statOff := di.di_5.bits[2]._inversed,
           cmdOn:=od.do_1.bits[6], cmdOff:=od.do_1.bits[7],
           StrSw:= IM.nu2  );

  (*  ПНС Насос смазки *)
  fb_pns(statOn := di.di_5.bits[0].value, statOff := di.di_5.bits[0]._inversed,
           cmdOn:=od.do_1.bits[0], cmdOff:=od.do_1.bits[1],
           StrSw:= IM.pns  );

  (*  В1 АВОМ вентилятор охлаждения *)
  fb_v1_Avom(statOn := di.di_5.bits[3].value, statOff := di.di_5.bits[3]._inversed,
           cmdOn:=od.do_1.bits[8], cmdOff:=od.do_1.bits[9],
           StrSw:= IM.v1_Avom  );

  (*  В2 АВОМ вентилятор охлаждения *)
  fb_v2_Avom(statOn := di.di_5.bits[4].value, statOff := di.di_5.bits[4]._inversed,
           cmdOn:=od.do_1.bits[10], cmdOff:=od.do_1.bits[11],
           StrSw:= IM.v2_Avom  );

  (*  В3 АВОМ вентилятор охлаждения *)
  fb_v3_Avom(statOn := di.di_5.bits[5].value, statOff := di.di_5.bits[5]._inversed,
           cmdOn:=od.do_1.bits[12], cmdOff:=od.do_1.bits[13],
           StrSw:= IM.v3_Avom  );

  (*  В4 АВОМ вентилятор охлаждения *)
  fb_v4_Avom(statOn := di.di_5.bits[6].value, statOff := di.di_5.bits[6]._inversed,
           cmdOn:=od.do_1.bits[14], cmdOff:=od.do_1.bits[15],
           StrSw:= IM.v4_Avom  );

  (*  МВ масляный выключатель *)
  fb_mv(statOn := di.di_7.bits[0].value, statOff := di.di_20.bits[3].value,
           basketRolledin:= di.di_7.bits[2], basketRolledout:= di.di_7.bits[2],
           cmdOn:=od.do_4.bits[6] , cmdOff:=od.do_4.bits[7],
           StrSw:= IM.mv  );

  (* Тен коллектора *)
  fb_TEN_kollectora(statOn := di.di_10.bits[1].value, statOff := di.di_10.bits[1]._inversed,
           cmdOn:=od.do_2.bits[6], cmdOff:=od.do_2.bits[6],
           StrSw:= IM.TEN_kollectora  );

  (* Калорифер АВОМ *)
  fb_KaloriferAVOM(statOn := di.di_10.bits[2].value, statOff := di.di_10.bits[2]._inversed,
           cmdOn:=od.do_2.bits[0], cmdOff:=od.do_2.bits[1],
           StrSw:= IM.KaloriferAVOM  );

  (* ЦМН *)
  fb_CMN(statOn := di.di_10.bits[3].value, statOff := di.di_10.bits[3]._inversed,
           cmdOn:=od.do_2.bits[4], cmdOff:=od.do_2.bits[5],
           StrSw:= IM.CMN);

  (* Тен маслобака *)
  fb_TEN_MB(statOn := di.di_10.bits[0].value, statOff := di.di_10.bits[0]._inversed,
           cmdOn:=od.do_2.bits[2], cmdOff:=od.do_2.bits[3],
           StrSw:= IM.TEN_MB);
  (*************************************************** singleSignals ********************************************)

  (* Перепад давления масло газ м*)
  fb_dP_maslo_gaz_Less100(signal :=di.di_20.bits[6], str_SS := IM.SingleSignals.dP_maslo_gaz_Less100);

  (* Перепад давления кран 1 *)
  fb_dp_kran1_Less100(signal :=di.di_4.bits[1], str_SS := IM.SingleSignals.dp_kran1_Less100);

  (* Неисправность цепей управления возбудителя *)
  fb_Vozbud_neispr_tsepey_upr_AVR_pit(signal :=di.di_6.bits[4], str_SS := IM.SingleSignals.Vozbud_neispr_tsepey_upr_AVR_pit);

  (* Возбудитель готовность *)
  fb_Vozbud_gotovnost(signal :=di.di_6.bits[0], str_SS := IM.SingleSignals.Vozbud_gotovnost);

  (* Возбудитель неисправность *)
  fb_Vozbud_neispravnost(signal :=di.di_21.bits[7], str_SS := IM.SingleSignals.Vozbud_neispravnost);

  (* ЩАВР 1 в работе *)
  fb_SHAVR1_v_rabote(signal :=di.di_13.bits[6], str_SS := IM.SingleSignals.SHAVR1_v_rabote);

  (* ЩАВР 2 в работе *)
  fb_SHAVR2_v_rabote(signal :=di.di_13.bits[7], str_SS := IM.SingleSignals.SHAVR2_v_rabote);

  (* ЩАВР 2 в работе *)
  fb_Avariinoe_otkluch_vikluchatelya(signal :=di.di_8.bits[0], str_SS := IM.SingleSignals.Avariinoe_otkluch_vikluchatelya);

  (* ЩАВР 2 в работе *)
  fb_Assinhronnii_hod_peregruzka(signal :=di.di_8.bits[1], str_SS := IM.SingleSignals.Assinhronnii_hod_peregruzka);

  (* ЩАВР 2 в работе *)
  fb_SHU_v_GPA_vkluch(signal :=di.di_8.bits[2], str_SS := IM.SingleSignals.SHU_v_GPA_vkluch);

  (* ЩАВР 2 в работе *)
  fb_SHP_v_GPA_vkluch(signal :=di.di_8.bits[3], str_SS := IM.SingleSignals.SHP_v_GPA_vkluch);

  (* ЩАВР 2 в работе *)
  fb_Uroven_masla_akkum(signal :=di.di_4.bits[2], str_SS := IM.SingleSignals.Uroven_masla_akkum);

  (* ЩАВР 2 в работе *)
  fb_NKU1_GPA_on(signal :=di.di_10.bits[4], str_SS := IM.SingleSignals.NKU1_GPA_on);

  (* ЩАВР 2 в работе *)
  fb_NKU2_GPA_on(signal :=di.di_10.bits[5], str_SS := IM.SingleSignals.NKU2_GPA_on);

  (* ЩАВР 2 в работе *)
  fb_AO_KC_ot_SHKS(signal :=di.di_20.bits[0], str_SS := IM.SingleSignals.AO_KC_ot_SHKS);

  (* ЩАВР 2 в работе *)
  fb_AO_GPA_ot_SHU(signal :=di.di_21.bits[2], str_SS := IM.SingleSignals.AO_GPA_ot_SHU);

  (* ЩАВР 2 в работе *)
  fb_BEAO_srabotal(signal :=di.di_18.bits[1], str_SS := IM.SingleSignals.BEAO_srabotal);

  (* ЩАВР 2 в работе *)
  fb_Chastotny_pusk(signal :=di.di_9.bits[0], str_SS := IM.SingleSignals.Chastotny_pusk);

  (* ЩАВР 2 в работе *)
  fb_Neuspesh_chastotny_pusk(signal :=di.di_9.bits[1], str_SS := IM.SingleSignals.Neuspesh_chastotny_pusk);

  (* ЩАВР 2 в работе *)
  fb_Rezhim_ruchnogo_regulirovaniya(signal :=di.di_9.bits[2], str_SS := IM.SingleSignals.Rezhim_ruchnogo_regulirovaniya);

  (* ЩАВР 2 в работе *)
  fb_Razreshenie_zagruzki_dvig(signal :=di.di_6.bits[1], str_SS := IM.SingleSignals.Razreshenie_zagruzki_dvig);

  (* ЩАВР 2 в работе *)
  fb_Osnovnoy_regul_off(signal :=di.di_6.bits[3], str_SS := IM.SingleSignals.Osnovnoy_regul_off);

  (* ЩАВР 2 в работе *)
  fb_Voltage_sekcii_norm(signal :=di.di_8.bits[4], str_SS := IM.SingleSignals.Voltage_sekcii_norm);

  (* ЩАВР 2 в работе *)
  fb_Reactorny_pusk(signal :=di.di_8.bits[5], str_SS := IM.SingleSignals.Reactorny_pusk);

  (* ЩАВР 2 в работе *)
  fb_NO_GPA_ot_SHU(signal :=di.di_21.bits[1], str_SS := IM.SingleSignals.NO_GPA_ot_SHU);

  (* ЩАВР 2 в работе *)
  fb_AO_GPA_ot_PRU(signal :=di.di_21.bits[3], str_SS := IM.SingleSignals.AO_GPA_ot_PRU);

  (* ЩАВР 2 в работе *)
  fb_Nalichie_BP1(signal :=di.di_11.bits[0], str_SS := IM.SingleSignals.Nalichie_BP1);

  (* ЩАВР 2 в работе *)
  fb_Nalichie_BP2(signal :=di.di_11.bits[1], str_SS := IM.SingleSignals.Nalichie_BP2);

  (* ЩАВР 2 в работе *)
  fb_Nalichie_BP3(signal :=di.di_11.bits[2], str_SS := IM.SingleSignals.Nalichie_BP3);

  (* ЩАВР 2 в работе *)
  fb_Nalichie_BP4(signal :=di.di_11.bits[3], str_SS := IM.SingleSignals.Nalichie_BP4);

  (* ЩАВР 2 в работе *)
  fb_Nalichie_BP5(signal :=di.di_11.bits[4], str_SS := IM.SingleSignals.Nalichie_BP5);

  (* ЩАВР 2 в работе *)
  fb_Nalichie_BP6(signal :=di.di_11.bits[5], str_SS := IM.SingleSignals.Nalichie_BP6);

  (* ЩАВР 2 в работе *)
  fb_Nalichie_BP7_BP8(signal :=di.di_11.bits[6], str_SS := IM.SingleSignals.Nalichie_BP7_BP8);

  (* ЩАВР 2 в работе *)
  fb_Nalichie_BP9_BP10(signal :=di.di_11.bits[7], str_SS := IM.SingleSignals.Nalichie_BP9_BP10);

  (* ЩАВР 2 в работе *)
  fb_Nalichie_cepei_upravlen_mv(signal :=di.di_12.bits[0], str_SS := IM.SingleSignals.Nalichie_cepei_upravlen_mv);

  (* ЩАВР 2 в работе *)
  fb_Nalichie_220BEAO(signal :=di.di_12.bits[1], str_SS := IM.SingleSignals.Nalichie_220BEAO);

  (* ЩАВР 2 в работе *)
  fb_Nalichie_per_220_na_vhode(signal :=di.di_12.bits[2], str_SS := IM.SingleSignals.Nalichie_per_220_na_vhode);

  (* ЩАВР 2 в работе *)
  fb_Nalichie_post_220_na_vhode(signal :=di.di_12.bits[3], str_SS := IM.SingleSignals.Nalichie_post_220_na_vhode);

  (* ЩАВР 2 в работе *)
  fb_Nalichie_BP11(signal :=di.di_12.bits[4], str_SS := IM.SingleSignals.Nalichie_BP11);

  (* ЩАВР 2 в работе *)
  fb_Nalichie_BP12(signal :=di.di_12.bits[4], str_SS := IM.SingleSignals.Nalichie_BP12);

  (* ЩАВР 2 в работе *)
  fb_Dver_SHU_pered_otkrita(signal :=di.di_13.bits[0], str_SS := IM.SingleSignals.Dver_SHU_pered_otkrita);

  (* ЩАВР 2 в работе *)
  fb_Dver_SHU_zad_otkrita(signal :=di.di_13.bits[1], str_SS := IM.SingleSignals.Dver_SHU_zad_otkrita);

  (* ЩАВР 2 в работе *)
  fb_EO_GPA_ot_knopki_SHU(signal :=di.di_14.bits[0], str_SS := IM.SingleSignals.EO_GPA_ot_knopki_SHU);

  (* ЩАВР 2 в работе *)
  fb_EO_EGPA_ot_PRY(signal :=di.di_14.bits[1], str_SS := IM.SingleSignals.EO_EGPA_ot_PRY);

  (* ЩАВР 2 в работе *)
  fb_Synchroniz_rezhima_K1(signal :=di.di_3.bits[4], str_SS := IM.SingleSignals.Synchroniz_rezhima_K1);

  (* ЩАВР 2 в работе *)
  fb_Potok_ms_posle_AVOM(signal :=di.di_3.bits[4], str_SS := IM.SingleSignals.Potok_ms_posle_AVOM);

    (* Выключатель основного ввода питания QF1  в положении включен   *)
  fb_QF1_on(signal :=di.di_7.bits[6], str_SS := IM.SingleSignals.QF1_on);

    (* Выключатель резервного ввода питания QF2  в положении включен   *)
  fb_QF2_on(signal :=di.di_7.bits[7], str_SS := IM.SingleSignals.QF2_on);

    (* Выключатель питания кранов:  QF23 110 В в положении включен   *)
  fb_QF23_on(signal :=di.di_8.bits[0], str_SS := IM.SingleSignals.QF23_on);

    (* Выключатели группы 1: QF4, QF5 в положении включен   *)
  fb_QF4_QF5_on(signal :=di.di_8.bits[1], str_SS := IM.SingleSignals.QF4_QF5_on);

    (* Выключатели группы 2: QF6, QF7 в положении включен   *)
  fb_QF6_QF7_on(signal :=di.di_8.bits[2], str_SS := IM.SingleSignals.QF6_QF7_on);

    (* Выключатели группы 3: QF8, QF9 в положении включен   *)
  fb_QF8_QF9_on(signal :=di.di_8.bits[3], str_SS := IM.SingleSignals.QF8_QF9_on);

    (* Выключатели группы 4: QF10, QF11 в положении включен   *)
  fb_QF10_QF11_on(signal :=di.di_8.bits[4], str_SS := IM.SingleSignals.QF10_QF11_on);

    (* Выключатели группы 5: QF12, QF13 в положении включен   *)
  fb_QF12_QF13_on(signal :=di.di_8.bits[5], str_SS := IM.SingleSignals.QF12_QF13_on);

    (* Выключатели группы 6: QF14, QF15 в положении включен   *)
  fb_QF14_QF15_on(signal :=di.di_8.bits[6], str_SS := IM.SingleSignals.QF14_QF15_on);

    (* Выключатели группы : QF22 в положении включен   *)
  fb_QF22_on(signal :=di.di_14.bits[2], str_SS := IM.SingleSignals.QF22_on);

    (* Неисправность источников питания группы 1: G1, G2 (=24 В)   *)
  fb_NS_G1_G2(signal :=di.di_8.bits[7], str_SS := IM.SingleSignals.NS_G1_G2);

    (* Неисправность источников питания группы 2: G3, G4 (=24 В)   *)
  fb_NS_G3_G4(signal :=di.di_9.bits[0], str_SS := IM.SingleSignals.NS_G3_G4);

    (* Неисправность источников питания внутренних ПТС: G15, G16 (=24 В)   *)
  fb_NS_G15_G16(signal :=di.di_9.bits[1], str_SS := IM.SingleSignals.NS_G15_G16);

    (* Неисправность источника питания аналоговых сигналов: G17 (=24 В)   *)
  fb_NS_G17(signal :=di.di_9.bits[2], str_SS := IM.SingleSignals.NS_G17);

    (* Неисправность источников питания группы 3: G5, G6 (=24 В)   *)
  fb_NS_G5_G6(signal :=di.di_9.bits[3], str_SS := IM.SingleSignals.NS_G5_G6);

    (* Неисправность источников питания группы 4: G7, G8 (=24 В)   *)
  fb_NS_G7_G8(signal :=di.di_9.bits[4], str_SS := IM.SingleSignals.NS_G7_G8);

    (* Неисправность источников питания внешних цепей: G18, G19 (=24 В)   *)
  fb_NS_G18_G19(signal :=di.di_9.bits[5], str_SS := IM.SingleSignals.NS_G18_G19);

    (* Неисправность источников питания группы 5: G9, G10, G11, G12 (=110 В)   *)
  fb_NS_G10_G11(signal :=di.di_9.bits[6], str_SS := IM.SingleSignals.NS_G10_G11);

    (* Неисправность источников питания G13, G14 (=24 В)   *)
  fb_NS_G13_G14(signal :=di.di_9.bits[7], str_SS := IM.SingleSignals.NS_G13_G14);

  (*************************************************** SingleOutputs ********************************************)

  (* Идикация НО (подсветка кнопки на шкафу)   *)
  fb_Rabota_EGPA(str_SO := IM.SingleOutputs.Rabota_EGPA, signal:=od.do_4.bits[2]);

  (* Взвод включения БЭАО по неисправности ПТС   *)
  fb_Neispr_EGPA(str_SO := IM.SingleOutputs.Neispr_EGPA, signal:=od.do_4.bits[0]);

  (* Авария ЭГПА в КЦ
  fb_Avary_EGPA(str_SO := IM.SingleOutputs.Avary_EGPA, signal:=od.do_4.bits[1);  *)

  (* Сброс включения БЭАО по неисправности ПТС   *)
  fb_U_lamp_SHU(str_SO := IM.SingleOutputs.U_lamp_SHU, signal:=od.do_4.bits[3]);

  (* Индикация ПС Фонарь   *)
  fb_AO_knopka_ind(str_SO := IM.SingleOutputs.AO_knopka_ind, signal:=od.do_4.bits[4]);

  (* Индикация АС Фонарь   *)
  fb_Pusk(str_SO := IM.SingleOutputs.Pusk_SHUP, signal:=od.do_4.bits[8]);

  (* Отключение МВ1 от КНА   *)
  fb_Stop_SHUP(str_SO := IM.SingleOutputs.Stop_SHUP, signal:=od.do_4.bits[9]);

  (* Отключение МВ1 от КНА   *)
  fb_NO_fonar(str_SO := IM.SingleOutputs.NO_fonar, signal:=od.do_3.bits[10]);

  (* Отключение МВ1 от КНА   *)
  fb_PC_fonar(str_SO := IM.SingleOutputs.PC_fonar, signal:=od.do_3.bits[9]);

  (* Отключение МВ1 от КНА   *)
  fb_AC_fonar(str_SO := IM.SingleOutputs.AC_fonar, signal:=od.do_3.bits[8]);

  (* Отключение МВ1 от КНА   *)
  fb_Kr1_smazka(str_SO := IM.SingleOutputs.Kr1_smazka, signal:=od.do_0.bits[14]);

  (* Отключение МВ1 от КНА   *)
  fb_Kr2_smazka(str_SO := IM.SingleOutputs.Kr2_smazka, signal:=od.do_0.bits[15]);

  (* Отключение МВ1 от КНА   *)
  fb_Kr4_open_from_alg(str_SO := IM.SingleOutputs.Kr4_open_from_alg, signal:=od.do_0.bits[8]);

  (* Отключение МВ1 от КНА   *)
  fb_Synch_rej_K1(str_SO := IM.SingleOutputs.Synch_rej_K1, signal:=od.do_3.bits[13]);

   (**************************************** Аналоговые и Дискретные параметры ***********************************)
END_FUNCTION_BLOCK

FUNCTION_BLOCK proc_DO_Init
  VAR_INPUT
    init : BOOL;
  END_VAR
  VAR
    stDO_Ini : fb_DO_Init;
    inits : UINT;
  END_VAR
  VAR_INPUT
    initiales : UINT;
  END_VAR
  VAR_EXTERNAL
    od : DOconfig;
  END_VAR

  (* Инициализация начало. Входные дискретные параметры *)

  inits := 0; (* Флаг необходимости инициализации структур-дескрипторов *)

  (* Модуль A1-15 *)
  stDO_Ini(data_Ini := true, imit:=FALSE, strDO := od.do_0);
  inits := inits + BOOL_TO_UINT(stDO_Ini.Init);

  (* Модуль A1-16 *)
  stDO_Ini(data_Ini := true, imit:=FALSE, strDO := od.do_1);
  inits := inits + BOOL_TO_UINT(stDO_Ini.Init);

  (* Модуль A1-17 *)
  stDO_Ini(data_Ini := true, imit:=FALSE, strDO := od.do_2);
  inits := inits + BOOL_TO_UINT(stDO_Ini.Init);

  (* Модуль A1-18 *)
  stDO_Ini(data_Ini := true, imit:=FALSE, strDO := od.do_3);
  inits := inits + BOOL_TO_UINT(stDO_Ini.Init);

  (* Модуль A1-19 *)
  stDO_Ini(data_Ini := true, imit:=FALSE, strDO := od.do_4);
  inits := inits + BOOL_TO_UINT(stDO_Ini.Init);

  (* Модуль A1-23 *)
  stDO_Ini(data_Ini := true, imit:=FALSE, strDO := od.gpio_out);
  inits := inits + BOOL_TO_UINT(stDO_Ini.Init);
  initiales := 0;

  IF init THEN initiales := inits; END_IF;
END_FUNCTION_BLOCK

FUNCTION_BLOCK fb_ph_CustomPhase
  VAR_INPUT
    PhaseNumber : UINT;
  END_VAR
  VAR_IN_OUT
    StrPh : struct_PhaseAlgoritm;
  END_VAR
  VAR
    CommandFault_Trig : R_TRIG;
    reset_Trig : R_TRIG;
    _statusDualInput : TYPE_statusDualInput;
  END_VAR

  IF StrPh.run AND NOT StrPh.start THEN
  	StrPh.start := TRUE;
  	StrPh.top := FALSE;
  	StrPh.error := FALSE;
            StrPh.run:=FALSE;
  END_IF;

  IF StrPh.top THEN StrPh.error := FALSE; END_IF;

  reset_Trig(CLK := StrPh.reset);
  IF reset_Trig.Q THEN
  	StrPh.start := FALSE;
  	StrPh.error := FALSE;
  	StrPh.top := FALSE;
            StrPh.run:=FALSE;
            StrPh.reset:=FALSE;
  END_IF;

  StrPh.startStatus := SHL(BOOL_TO_DWORD(StrPh.start), PhaseNumber);
  StrPh.errorStatus := SHL(BOOL_TO_DWORD(StrPh.error), PhaseNumber);
  StrPh.topStatus := SHL(BOOL_TO_DWORD(StrPh.top), PhaseNumber);
END_FUNCTION_BLOCK

FUNCTION_BLOCK fb_DOSourceMlp
  VAR_IN_OUT
    arDout : TWordData;
  END_VAR
  VAR_INPUT
    err_mod : TItemDIN;
  END_VAR
  VAR_IN_OUT
    strDO : struct_DO;
  END_VAR
  VAR
    bitNumber : INT;
  END_VAR

  strDO.blConnect := ((UINT_TO_WORD(err_mod.wValue) = 20) and (UINT_TO_WORD(err_mod.wFlags) = 192));

  strDO.value:=0;

  FOR bitNumber:=0 TO 15 BY 1 DO
  	strDO.value:=strDO.value OR (SHL(BOOL_TO_WORD(strDO.bits[bitNumber]),bitNumber));
  END_FOR;

  IF NOT strDO.imit THEN
  	 arDout.wValue:= WORD_TO_UINT(strDO.value);
  END_IF;
END_FUNCTION_BLOCK

FUNCTION_BLOCK fb_DI_Init
  VAR_INPUT
    data_Ini : BOOL;
    imit : BOOL      := FALSE;
  END_VAR
  VAR_IN_OUT
    strDI : struct_DI;
  END_VAR
  VAR_OUTPUT
    Init : BOOL      := FALSE;
  END_VAR

  (*****            Функциональный блок переинициализации структуры-дескриптора канала дискретного ввода        *****)

   Init := FALSE;

      IF data_Ini THEN                            (* Параметрам требуется переинициализация. *)
          strDI.imit       := imit;
          data_Ini:=FALSE;
          Init := TRUE;
      END_IF;
    IF Init THEN
  imit:=FALSE;
      END_IF;
END_FUNCTION_BLOCK

FUNCTION_BLOCK fb_AO_Init
  VAR_INPUT
    data_Ini : BOOL;
    outLL : LREAL      := 4000.0;
    outHL : LREAL      := 20000.0;
    newLL : LREAL;
    newHL : LREAL;
    newLL_ISVALIDREF : BOOL;
    newHL_ISVALIDREF : BOOL;
  END_VAR
  VAR_IN_OUT
    strAO : struct_AO;
  END_VAR
  VAR_OUTPUT
    Init : BOOL      := FALSE;
  END_VAR

  (*****            Функциональный блок переинициализации структуры-дескриптора канала аналогового ввода.            *****)

   Init := FALSE;

      IF data_Ini THEN                            (* Параметрам требуется переинициализация. *)
          strAO.outLL                := outLL;
          strAO.outHL                := outHL;
          strAO.newLL                := newLL;
          strAO.newHL                := newHL;
          strAO.newLL_ISVALIDREF     := newLL_ISVALIDREF;
          strAO.newHL_ISVALIDREF     := newHL_ISVALIDREF;
          data_Ini:=FALSE;
          Init := TRUE;
      END_IF;
   IF Init THEN
         (* outLL:=0.0;*)
         (* outHL:=0.0;*)
          newLL:=0.0;
          newHL:=0.0;
          newLL_ISVALIDREF:= FALSE;
          newHL_ISVALIDREF:= FALSE;
   END_IF;
END_FUNCTION_BLOCK

FUNCTION_BLOCK fb_AOSourceMlp
  VAR_IN_OUT
    OutCurrent : TDoubleData;
    strAO : struct_AO;
  END_VAR
  VAR
    _sunpackerCommand : fb_sunpackerCommand;
    source : BYTE;
    source_for_Status : BYTE;
    cmd : BYTE;
    cmd_for_Status : BYTE;
    lastCmd : BYTE;
    command_error_for_Status : BYTE;
    resetCmdTimer : TON;
    resetCmdTimerPriznak : BOOL;
    secondTack : BOOL;
    inOpcCommandsDisabled : BOOL;
  END_VAR
  VAR_INPUT RETAIN
    retainLL : LREAL;
    retainHL : LREAL;
  END_VAR

  IF NOT secondTack THEN
            IF (strAO.newLL <> retainLL) AND (retainLL <> 0.0) THEN  strAO.LL := retainLL;
            ELSE strAO.LL:= strAO.newLL; END_IF;
  	IF (strAO.newHL <> retainHL) AND (retainHL <> 0.0) THEN  strAO.HL := retainHL;
            ELSE strAO.HL:= strAO.newHL; END_IF;

  	secondTack  := FALSE;
  END_IF;
  strAO.blConnect :=(UINT_TO_WORD(OutCurrent.wFlags) AND 16#0040) <> 0;
  strAO.OpcCommandsDisabled := inOpcCommandsDisabled;

  _sunpackerCommand(command := strAO.inCommand);
  	source := _sunpackerCommand.source;
  	cmd := _sunpackerCommand.cmd;

  IF cmd <> 0 AND lastCmd <> cmd and (((NOT strAO.opcCommandsDisabled) AND source > 0) OR source = 0) then
  	CASE BYTE_TO_INT(cmd) OF
  	(*cmd_ChangeValue*) 1 : 	IF ((NOT strAO.newLL_ISVALIDREF) OR (strAO.nValue >= strAO.LL)) AND
                                             ((NOT strAO.newHL_ISVALIDREF) OR (strAO.nValue <= strAO.HL) ) THEN
  					strAO.Value := strAO.nValue;
  				END_IF;
  	(*cmd_ChangeLimits*) 2 : 	strAO.LL := strAO.newLL; retainLL:= strAO.LL;
  				strAO.HL := strAO.newHL; retainHL:= strAO.HL;
  	END_CASE;
  	source_for_Status := source;
  	cmd_for_Status := cmd;
  	command_error_for_Status := 0;
  	resetCmdTimer(IN := FALSE);
  	resetCmdTimerPriznak := TRUE;
  END_IF;
  lastCmd := cmd;

  IF (strAO.HL <> strAO.LL) THEN
  	OutCurrent.dblValue := ((strAO.Value - strAO.LL) * (strAO.outHL-strAO.outLL)/(strAO.HL - strAO.LL )) + strAO.outLL;
  END_IF;

  resetCmdTimer(IN := resetCmdTimerPriznak, PT := T#5S);
  IF resetCmdTimer.Q THEN
  	resetCmdTimerPriznak := FALSE;
  	source_for_Status := 0;
  	cmd_for_Status := 0;
  	command_error_for_Status := 0;
  END_IF;

  strAO.status := SHL(BYTE_TO_DWORD(source_for_Status), 29)
  			OR SHL(BYTE_TO_DWORD(cmd_for_Status), 26)
  			OR SHL(BYTE_TO_DWORD(command_error_for_Status), 23)
  			OR SHL(BOOL_TO_DWORD(strAO.OpcCommandsDisabled ), 21);
END_FUNCTION_BLOCK

FUNCTION_BLOCK proc_DO
  VAR
    do_0 : fb_DOSourceMlp;
    do_1 : fb_DOSourceMlp;
    do_2 : fb_DOSourceMlp;
    do_3 : fb_DOSourceMlp;
    do_4 : fb_DOSourceMlp;
    gpio_out : fb_DOSourceMlp;
  END_VAR
  VAR_EXTERNAL
    od : DOconfig;
    arDOUT_0 : TWordData;
    arDOUT_1 : TWordData;
    arDOUT_2 : TWordData;
    arDOUT_3 : TWordData;
    arDOUT_4 : TWordData;
    arERR_66 : TItemDIN;
    arDOUT_66 : TWordData;
    arERR_0 : TItemDIN;
    arERR_1 : TItemDIN;
    arERR_2 : TItemDIN;
    arERR_15 : TItemDIN;
    arERR_16 : TItemDIN;
    A1_1_err_mode : UINT;
    A1_2_err_mode : UINT;
    A1_3_err_mode : UINT;
    A2_1_err_mode : UINT;
    A2_4_err_mode : UINT;
    DO_0_wValue : UINT;
    DO_1_wValue : UINT;
    DO_2_wValue : UINT;
    DO_3_wValue : UINT;
    DO_4_wValue : UINT;
  END_VAR

  (* Циклический опрос. Входные дискретные параметры *)

  (* Модуль A1-1 *)
  do_0(arDout := arDOUT_0, strDO := od.do_0, err_mod:=arERR_0);
  DO_0_wValue:=arDOUT_0.wValue;
  A1_1_err_mode:= arERR_0.wValue;

  (* Модуль A1-2 *)
  do_1(arDout := arDOUT_1, strDO := od.do_1, err_mod:=arERR_1);
  DO_1_wValue:=arDOUT_1.wValue;
  A1_2_err_mode:= arERR_1.wValue;

  (* Модуль A1-3 *)
  do_2(arDout := arDOUT_2, strDO := od.do_2, err_mod:=arERR_2);
  DO_2_wValue:=arDOUT_2.wValue;
  A1_3_err_mode:= arERR_2.wValue;

  (* Модуль A2-1 *)
  do_3(arDout := arDOUT_3, strDO := od.do_3, err_mod:=arERR_15);
  DO_3_wValue:=arDOUT_3.wValue;
  A2_1_err_mode:= arERR_15.wValue;

  (* Модуль A2-1 *)
  do_4(arDout := arDOUT_4, strDO := od.do_4, err_mod:=arERR_15);
  DO_4_wValue:=arDOUT_4.wValue;
  A2_4_err_mode:= arERR_16.wValue;

  gpio_out(arDout := arDOUT_66, strDO := od.gpio_out, err_mod:=arERR_66);
END_FUNCTION_BLOCK

FUNCTION_BLOCK proc_DI_Init
  VAR_INPUT
    init : BOOL;
  END_VAR
  VAR
    stDI_Ini : fb_DI_Init;
    inits : UINT;
  END_VAR
  VAR_INPUT
    initiales : UINT;
  END_VAR
  VAR_EXTERNAL
    di : DiConfig;
  END_VAR

  (* Инициализация начало. Входные дискретные параметры *)

  inits := 0; (* Флаг необходимости инициализации структур-дескрипторов *)

  (* Модуль A1-1 *)

  stDI_Ini(data_Ini := true, imit:=FALSE, strDI := di.di_0);
  inits := inits + BOOL_TO_UINT(stDI_Ini.Init);

  stDI_Ini(data_Ini := true, imit:=FALSE, strDI := di.di_1);
  inits := inits + BOOL_TO_UINT(stDI_Ini.Init);

  (* Модуль A1-2 *)
  stDI_Ini(data_Ini := true, imit:=FALSE, strDI := di.di_2);
  inits := inits + BOOL_TO_UINT(stDI_Ini.Init);

  stDI_Ini(data_Ini := true, imit:=FALSE, strDI := di.di_3);
  inits := inits + BOOL_TO_UINT(stDI_Ini.Init);

  (* Модуль A1-3 *)
  stDI_Ini(data_Ini := true, imit:=FALSE, strDI := di.di_4);
  inits := inits + BOOL_TO_UINT(stDI_Ini.Init);

  stDI_Ini(data_Ini := true, imit:=FALSE, strDI := di.di_5);
  inits := inits + BOOL_TO_UINT(stDI_Ini.Init);

  (* Модуль A1-4 *)
  stDI_Ini(data_Ini := true, imit:=FALSE, strDI := di.di_6);
  inits := inits + BOOL_TO_UINT(stDI_Ini.Init);

  stDI_Ini(data_Ini := true, imit:=FALSE, strDI := di.di_7);
  inits := inits + BOOL_TO_UINT(stDI_Ini.Init);

  (* Модуль A1-5 *)
  stDI_Ini(data_Ini := true, imit:=FALSE,  strDI := di.di_8);
  inits := inits + BOOL_TO_UINT(stDI_Ini.Init);

  stDI_Ini(data_Ini := true, imit:=FALSE,  strDI := di.di_9);
  inits := inits + BOOL_TO_UINT(stDI_Ini.Init);

  (* Модуль A1-6 *)
  stDI_Ini(data_Ini := true, imit:=FALSE,  strDI := di.di_10);
  inits := inits + BOOL_TO_UINT(stDI_Ini.Init);

  stDI_Ini(data_Ini := true, imit:=FALSE,  strDI := di.di_11);
  inits := inits + BOOL_TO_UINT(stDI_Ini.Init);

  (* Модуль A1-7 *)
  stDI_Ini(data_Ini := true, imit:=FALSE, strDI := di.di_12);
  inits := inits + BOOL_TO_UINT(stDI_Ini.Init);

  stDI_Ini(data_Ini := true, imit:=FALSE, strDI := di.di_13);
  inits := inits + BOOL_TO_UINT(stDI_Ini.Init);

  (* Модуль A1-8 *)
  stDI_Ini(data_Ini := true, imit:=FALSE, strDI := di.di_14);
  inits := inits + BOOL_TO_UINT(stDI_Ini.Init);

  stDI_Ini(data_Ini := true, imit:=FALSE, strDI := di.di_16);
  inits := inits + BOOL_TO_UINT(stDI_Ini.Init);

  stDI_Ini(data_Ini := true, imit:=FALSE, strDI := di.di_17);
  inits := inits + BOOL_TO_UINT(stDI_Ini.Init);

  stDI_Ini(data_Ini := true, imit:=FALSE, strDI := di.di_18);
  inits := inits + BOOL_TO_UINT(stDI_Ini.Init);

  stDI_Ini(data_Ini := true, imit:=FALSE, strDI := di.di_19);
  inits := inits + BOOL_TO_UINT(stDI_Ini.Init);

  stDI_Ini(data_Ini := true, imit:=FALSE, strDI := di.di_20);
  inits := inits + BOOL_TO_UINT(stDI_Ini.Init);

  stDI_Ini(data_Ini := true, imit:=FALSE, strDI := di.di_21);
  inits := inits + BOOL_TO_UINT(stDI_Ini.Init);

  initiales := 0;
  IF init THEN initiales := inits; END_IF;
END_FUNCTION_BLOCK

FUNCTION_BLOCK fb_DiSourceMlp
  VAR_INPUT
    arDIN : TItemDIN;
    err_mod : TItemDIN;
  END_VAR
  VAR_IN_OUT
    strDI : struct_DI;
  END_VAR
  VAR_OUTPUT
    Bounce : BOOL;
  END_VAR
  VAR
    _value : WORD;
    _reliability : BOOL;
    bitNumber : INT;
    bitNum : INT;
  END_VAR

  strDI.blConnect := (*((UINT_TO_WORD(arDIN.wFlags) = 1472) and*) (UINT_TO_WORD(err_mod.wValue) = 20) and (UINT_TO_WORD(err_mod.wFlags) = 192);
  Bounce := (UINT_TO_WORD(arDIN.wFlags) AND 16#0020) <> 0;

  If NOT strDI.imit THEN
  _value:=UINT_TO_WORD(arDIN.wValue);

      IF strDI.blConnect THEN
            strDI.reliability:=0;
            strDI.value:=0;
  	FOR bitNumber:=0 TO 7 BY 1 DO

  		_reliability:=WORD_TO_BOOL(SHR(_value, bitNumber*2) AND 16#2);
  		strDI.reliability:=strDI.reliability OR SHL(BOOL_TO_WORD(_reliability),bitNumber);
  		IF _reliability THEN
  			strDI.value:=strDI.value OR SHL((SHR(_value, bitNumber*2) AND 16#1),bitNumber);
  		END_IF;
  	END_FOR;
      ELSE
  	strDI.reliability := 0;
      END_IF;

      FOR bitNum:=0 TO 15 BY 1 DO
  	          strDI.bits[bitNum].reliability :=WORD_TO_BOOL(SHR(strDI.reliability, bitNum) AND 16#1);
  	IF strDI.bits[bitNum].reliability THEN
  		strDI.bits[bitNum].value :=WORD_TO_BOOL(SHR(strDI.value, bitNum) AND 16#1);
                      strDI.bits[bitNum]._inversed :=NOT strDI.bits[bitNum].value;
  	END_IF;
      END_FOR;

  END_IF;
END_FUNCTION_BLOCK

FUNCTION TwoUint_To_UDINT : UDINT
  VAR_INPUT
    val1 : UINT;
    val2 : UINT;
  END_VAR

  TwoUint_To_UDINT:= DWORD_TO_UDINT(UINT_TO_DWORD(val1) OR shl(UINT_TO_DWORD(val2), 16));
END_FUNCTION

FUNCTION_BLOCK proc_DI
  VAR
    di_0 : fb_DiSourceMlp;
    di_1 : fb_DiSourceMlp;
    di_2 : fb_DiSourceMlp;
    di_3 : fb_DiSourceMlp;
    di_4 : fb_DiSourceMlp;
    di_5 : fb_DiSourceMlp;
    di_6 : fb_DiSourceMlp;
    di_7 : fb_DiSourceMlp;
    di_8 : fb_DiSourceMlp;
    di_9 : fb_DiSourceMlp;
    di_10 : fb_DiSourceMlp;
    di_11 : fb_DiSourceMlp;
    di_12 : fb_DiSourceMlp;
    di_13 : fb_DiSourceMlp;
    di_14 : fb_DiSourceMlp;
    di_15 : fb_DiSourceMlp;
    di_16 : fb_DiSourceMlp;
    di_17 : fb_DiSourceMlp;
    di_18 : fb_DiSourceMlp;
    di_19 : fb_DiSourceMlp;
    di_20 : fb_DiSourceMlp;
    di_21 : fb_DiSourceMlp;
  END_VAR
  VAR_EXTERNAL
    arDIN_0 : TItemDIN;
    arDIN_1 : TItemDIN;
    arDIN_2 : TItemDIN;
    arDIN_3 : TItemDIN;
    arDIN_4 : TItemDIN;
    arDIN_5 : TItemDIN;
    arDIN_6 : TItemDIN;
    arDIN_7 : TItemDIN;
    arDIN_8 : TItemDIN;
    arDIN_9 : TItemDIN;
    arDIN_10 : TItemDIN;
    arDIN_11 : TItemDIN;
    arDIN_12 : TItemDIN;
    arDIN_13 : TItemDIN;
    arDIN_14 : TItemDIN;
    arDIN_15 : TItemDIN;
    arDIN_16 : TItemDIN;
    arDIN_17 : TItemDIN;
    arDIN_18 : TItemDIN;
    arDIN_19 : TItemDIN;
    arDIN_20 : TItemDIN;
    arDIN_21 : TItemDIN;
    di : DiConfig;
    DI_0_1_wValue : UDINT;
    DI_10_11_wValue : UDINT;
    DI_12_13_wValue : UDINT;
    DI_14_15_wValue : UDINT;
    DI_16_17_wValue : UDINT;
    DI_18_19_wValue : UDINT;
    DI_20_21_wValue : UDINT;
    DI_2_3_wValue : UDINT;
    DI_4_5_wValue : UDINT;
    DI_6_7_wValue : UDINT;
    DI_8_9_wValue : UDINT;
    A1_12_err_mode : UINT;
    A1_13_err_mode : UINT;
    A1_14_err_mode : UINT;
    A1_15_err_mode : UINT;
    A2_10_err_mode : UINT;
    A2_4_err_mode : UINT;
    A2_5_err_mode : UINT;
    A2_6_err_mode : UINT;
    A2_7_err_mode : UINT;
    A2_8_err_mode : UINT;
    A2_9_err_mode : UINT;
    arERR_11 : TItemDIN;
    arERR_12 : TItemDIN;
    arERR_13 : TItemDIN;
    arERR_14 : TItemDIN;
    arERR_18 : TItemDIN;
    arERR_19 : TItemDIN;
    arERR_20 : TItemDIN;
    arERR_21 : TItemDIN;
    arERR_22 : TItemDIN;
    arERR_23 : TItemDIN;
    arERR_24 : TItemDIN;
  END_VAR

  (* Циклический опрос. Входные дискретные параметры *)
  (* Модуль A1-12 *)
  di_0(arDIN := arDIN_0, strDI:=di.di_0, err_mod:=arERR_11);
  di_1(arDIN := arDIN_1, strDI:=di.di_1, err_mod:=arERR_11);
  DI_0_1_wValue:=TwoUint_To_UDINT(arDIN_0.wValue, arDIN_1.wValue);
  A1_12_err_mode:= arERR_11.wValue;

  (* Модуль A1-13 *)
  di_2(arDIN := arDIN_2, strDI:=di.di_2,  err_mod:=arERR_12);
  di_3(arDIN := arDIN_3, strDI:=di.di_3,  err_mod:=arERR_12);
  DI_2_3_wValue:=TwoUint_To_UDINT(arDIN_2.wValue, arDIN_3.wValue);
  A1_13_err_mode:= arERR_12.wValue;

  (* Модуль A1-14 *)
  di_4(arDIN := arDIN_4, strDI:=di.di_4,  err_mod:=arERR_13);
  di_5(arDIN := arDIN_5, strDI:=di.di_5,  err_mod:=arERR_13);
  DI_4_5_wValue:=TwoUint_To_UDINT(arDIN_4.wValue, arDIN_5.wValue);
  A1_14_err_mode:= arERR_13.wValue;

  (* Модуль A1-15 *)
  di_6(arDIN := arDIN_6, strDI:=di.di_6,  err_mod:=arERR_14);
  di_7(arDIN := arDIN_7, strDI:=di.di_7,  err_mod:=arERR_14);
  DI_6_7_wValue:=TwoUint_To_UDINT(arDIN_6.wValue, arDIN_7.wValue);
  A1_15_err_mode:= arERR_14.wValue;

  (* Модуль A2-4 *)
  di_8(arDIN := arDIN_8, strDI:=di.di_8,  err_mod:=arERR_18);
  di_9(arDIN := arDIN_9, strDI:=di.di_9,  err_mod:=arERR_18);
  DI_8_9_wValue:=TwoUint_To_UDINT(arDIN_8.wValue, arDIN_9.wValue);
  A2_4_err_mode:= arERR_18.wValue;

  (* Модуль A2-5 *)
  di_10(arDIN := arDIN_10, strDI:=di.di_10,  err_mod:=arERR_19);
  di_11(arDIN := arDIN_11, strDI:=di.di_11,  err_mod:=arERR_19);
  DI_10_11_wValue:=TwoUint_To_UDINT(arDIN_10.wValue, arDIN_11.wValue);
  A2_5_err_mode:= arERR_19.wValue;

  (* Модуль A2-6 *)
  di_12(arDIN := arDIN_12, strDI:=di.di_12,  err_mod:=arERR_20);
  di_13(arDIN := arDIN_13, strDI:=di.di_13,  err_mod:=arERR_20);
  DI_12_13_wValue:=TwoUint_To_UDINT(arDIN_12.wValue, arDIN_13.wValue);
  A2_6_err_mode:= arERR_20.wValue;

  (* Модуль A2-7 *)
  di_14(arDIN := arDIN_14, strDI:=di.di_14,  err_mod:=arERR_21);
  di_15(arDIN := arDIN_15, strDI:=di.di_15,  err_mod:=arERR_21);
  DI_14_15_wValue:=TwoUint_To_UDINT(arDIN_14.wValue, arDIN_15.wValue);
  A2_7_err_mode:= arERR_21.wValue;

  di_16(arDIN := arDIN_16, strDI:=di.di_16,  err_mod:=arERR_22);
  di_17(arDIN := arDIN_17, strDI:=di.di_17,  err_mod:=arERR_22);
  DI_16_17_wValue:=TwoUint_To_UDINT(arDIN_16.wValue, arDIN_17.wValue);
  A2_8_err_mode:= arERR_22.wValue;

  di_18(arDIN := arDIN_18, strDI:=di.di_18,  err_mod:=arERR_23);
  di_19(arDIN := arDIN_19, strDI:=di.di_19,  err_mod:=arERR_23);
  DI_18_19_wValue:=TwoUint_To_UDINT(arDIN_18.wValue, arDIN_19.wValue);
  A2_9_err_mode:= arERR_23.wValue;

  di_20(arDIN := arDIN_20, strDI:=di.di_20,  err_mod:=arERR_24);
  di_21(arDIN := arDIN_21, strDI:=di.di_21,  err_mod:=arERR_24);
  DI_20_21_wValue:=TwoUint_To_UDINT(arDIN_20.wValue, arDIN_21.wValue);
  A2_10_err_mode:= arERR_24.wValue;
END_FUNCTION_BLOCK

FUNCTION_BLOCK proc_AO_Init
  VAR_INPUT
    init : BOOL;
  END_VAR
  VAR
    stAO_Ini : fb_AO_Init;
    inits : UINT;
  END_VAR
  VAR_INPUT
    initiales : UINT;
  END_VAR
  VAR_EXTERNAL
    ao : AOConfig;
  END_VAR

  (* Инициализация начало. Входные аналоговые параметры *)

  inits := 0; (* Флаг необходимости инициализации структур-дескрипторов *)

  (* Модуль A10 *)
  (* [A10, AO0] Резерв (A) *)
  stAO_Ini(data_Ini := TRUE, (*outLL := 4000.0, outHL := 20000.0,*)
    newLL_ISVALIDREF := TRUE, newHL_ISVALIDREF := TRUE,
    newLL := 0.0, newHL := 100.0,
    strAO := ao.Reserv_AO_1);
  inits := inits + BOOL_TO_UINT(stAO_Ini.Init);

  (* [A1-10, AO1] Резерв (A) *)
  stAO_Ini(data_Ini := TRUE, (*outLL := 4000.0, outHL := 20000.0,*)
    (*newLL_ISVALIDREF := TRUE, newHL_ISVALIDREF := TRUE,*)
    (*newLL := 0.0, newHL := 100.0,*)
  strAO := ao.Reserv_AO_2);
  inits := inits + BOOL_TO_UINT(stAO_Ini.Init);

  initiales := 0;
  IF init THEN initiales := inits; END_IF;
END_FUNCTION_BLOCK

FUNCTION_BLOCK fb_Timings
  VAR_EXTERNAL CONSTANT
    req_Cycle : REAL;
  END_VAR
  VAR_EXTERNAL
    gF_T_100mSec : BOOL;
    gT_1Sec : BOOL;
    gF_T_1Sec : BOOL;
    gT_1Min : BOOL;
    gR_T_1Min : BOOL;
    gF_T_1Min : BOOL;
    del_T : REAL;
    cur_Cycle : REAL;
  END_VAR
  VAR
    Tmr_100_ms : REAL;
  END_VAR
  VAR_EXTERNAL
    T_1SEC : REAL;
  END_VAR
  VAR
    Tmr_1_s : REAL;
    Tmr_1_min : REAL;
  END_VAR

  (* Обработка времени. *)
  Tmr_100_ms := Tmr_100_ms + cur_Cycle;
  gF_T_100mSec := FALSE;
  IF Tmr_100_ms >= 0.1 THEN Tmr_100_ms := 0.0; gF_T_100mSec := TRUE; END_IF;

  Tmr_1_s := Tmr_1_s + cur_Cycle;
  gF_T_1Sec := FALSE;
  IF Tmr_1_s >= 1.0 THEN Tmr_1_s := 0.0; gF_T_1Sec := TRUE; END_IF;

  T_1SEC := T_1SEC + cur_Cycle;
  gT_1Sec := FALSE;
  IF T_1SEC >= 2.0 THEN T_1SEC := 0.0;
    ELSIF T_1SEC >= 1.0 THEN gT_1Sec := TRUE; END_IF;

  IF Tmr_1_min > 60.0 THEN
      Tmr_1_min := 0.0; gF_T_1Min := gT_1Min; gT_1Min := NOT gT_1Min; gR_T_1Min := gT_1Min;
    ELSE
      Tmr_1_min := Tmr_1_min + cur_Cycle; gR_T_1Min := FALSE; gF_T_1Min := FALSE;
  END_IF;
  del_T:= cur_Cycle;
END_FUNCTION_BLOCK

FUNCTION_BLOCK fb_ph_DIprotection
  VAR_IN_OUT
    StrDiP : struct_DiProtection;
  END_VAR
  VAR_INPUT
    act : TYPE_PhaseAlgoritmAction;
    PhaseNumber : UINT;
  END_VAR
  VAR_IN_OUT
    StrPh : struct_PhaseAlgoritm;
  END_VAR
  VAR
    CommandFault_Trig : R_TRIG;
    reset_Trig : R_TRIG;
    _statusDualInput : TYPE_statusDualInput;
  END_VAR

  IF StrPh.run AND NOT StrPh.start THEN
  	StrPh.start := TRUE;
  	StrPh.top := FALSE;
  	StrPh.error := FALSE;
            StrPh.run:=FALSE;

  	CASE act OF
  		(*PhaseAlgoritmAction.run*)    _run : runDiProtection(StrDiP); (*cmd_run*)
  		(*PhaseAlgoritmAction.reset*)_reset : resetDiProtection(StrDiP); (*cmd_reset*)
  	END_CASE;
  END_IF;

  IF StrPh.start AND NOT StrPh.top THEN
                      CommandFault_Trig(CLK := StrDiP.hasError);
                      IF CommandFault_Trig.Q THEN
  	          StrPh.error := TRUE;
                      END_IF;

  		CASE act OF
  		(*PhaseAlgoritmAction.run*)    _run:    StrPh.top:=StrDiP.isRunning;

  		(*PhaseAlgoritmAction.reset*) _reset:   StrPh.top := NOT StrDiP.isRunning;
  		END_CASE;

  END_IF;

  IF StrPh.top THEN
  StrPh.error := FALSE;
  END_IF;

  reset_Trig(CLK := StrPh.reset);
  IF reset_Trig.Q THEN
            StrPh.start := FALSE;
  	StrPh.error := FALSE;
  	StrPh.top := FALSE;
            StrPh.run:=FALSE;
            StrPh.reset:=FALSE;
  END_IF;

  StrPh.startStatus := SHL(BOOL_TO_DWORD(StrPh.start), PhaseNumber);
  StrPh.errorStatus := SHL(BOOL_TO_DWORD(StrPh.error), PhaseNumber);
  StrPh.topStatus := SHL(BOOL_TO_DWORD(StrPh.top), PhaseNumber);
END_FUNCTION_BLOCK

FUNCTION_BLOCK fb_DiscretParametr
  VAR_IN_OUT
    StrDP : struct_DiscretParametr;
  END_VAR
  VAR
    _sunpackerCommand : fb_sunpackerCommand;
    source : BYTE;
    cmd : BYTE;
    parametr : BYTE;
    lastParametr : BYTE;
    source_for_Status : BYTE;
    cmd_for_Status : BYTE;
    command_error_for_Status : BYTE;
    resetCmdTimer : TON;
    resetCmdTimerPriznak : BOOL;
    secondTact : BOOL;
  END_VAR

  IF NOT secondTact THEN
  	StrDP.Value := StrDP.currentValue;
  	secondTact := true;
  END_IF;

  StrDP.OpcCommandsDisabled := StrDP.inOpcCommandsDisabled;

  (* ---- Если управление с ВУ заблокировано, то передаем команду из алгоритма ---- *)
  IF StrDP.inOpcCommandsDisabled THEN
  	StrDP.inCommand := StrDP.inCommand_Alg;
  ELSE (* иначе передаем команду с АРМа*)
  	StrDP.inCommand := StrDP.inCommand_ARM;
  END_IF;

  _sunpackerCommand(command := StrDP.inCommand);
  	source := _sunpackerCommand.source;
            parametr := _sunpackerCommand.parametr;
  	cmd := _sunpackerCommand.cmd;

  IF NOT StrDP.inOpcCommandsDisabled THEN
  StrDP.newValue:= BYTE_TO_UINT(parametr);
  END_IF;

  IF cmd <> 0 AND StrDP.Value <> StrDP.newValue AND (((NOT StrDP.opcCommandsDisabled) AND source > 0) OR source = 0) then
  	CASE BYTE_TO_INT(cmd) OF
  	(*cmd_ChangeValue*) 1 :
                                    StrDP.Value := StrDP.newValue;
                                    StrDP.opcCommandsDisabled:=FALSE;
  	END_CASE;
  	source_for_Status := source;
  	cmd_for_Status := cmd;
  	resetCmdTimer(IN := FALSE);
  	resetCmdTimerPriznak := TRUE;
  END_IF;

  lastParametr := parametr;

  StrDP.status := SHL(BYTE_TO_DWORD(source_for_Status), 29)
  			OR SHL(BYTE_TO_DWORD(cmd_for_Status), 26)
  			OR SHL(BYTE_TO_DWORD(command_error_for_Status), 23)
  			OR SHL(BOOL_TO_DWORD(StrDP.OpcCommandsDisabled ), 21)
                                OR SHL(UINT_TO_DWORD(StrDP.Value), 5);

  resetCmdTimer(IN := resetCmdTimerPriznak, PT := T#5S);
  IF resetCmdTimer.Q THEN
  	resetCmdTimerPriznak := FALSE;
  	source_for_Status := 0;
  	cmd_for_Status := 0;
  	command_error_for_Status := 0;
  END_IF;
END_FUNCTION_BLOCK

FUNCTION_BLOCK fb_AI_Init
  VAR_INPUT
    data_Ini : BOOL;
    dLL : LREAL;
    dHL : LREAL;
    dLA : LREAL;
    dHA : LREAL;
    dLW : LREAL;
    dHW : LREAL;
    ISVALIDREF_LA : BOOL      := False;
    ISVALIDREF_HA : BOOL      := False;
    ISVALIDREF_LW : BOOL      := False;
    ISVALIDREF_HW : BOOL      := False;
    delayLA : TIME      := T#0S;
    delayLW : TIME      := T#0S;
    delayHW : TIME      := T#0S;
    delayHA : TIME      := T#0S;
    inpLL : LREAL      := 4000.0;
    inpHL : LREAL      := 20000.0;
    CurrentShotCircuit : LREAL      := 21000.0;
    CurrentBreakCircuit : LREAL      := 3700.0;
    dMaxChangeSpeed : LREAL;
    dMaxChangeSpeedDown : LREAL;
    histeresis : LREAL;
    aperturFilter : LREAL;
    exponentialFilter : LREAL;
    rassoglasovanie : LREAL;
    inOpcCommandsDisabled : BOOL;
  END_VAR
  VAR_IN_OUT
    strAI : struct_AI;
  END_VAR
  VAR_OUTPUT
    Init : BOOL      := FALSE;
  END_VAR

  (*****            Функциональный блок переинициализации структуры-дескриптора канала аналогового ввода.            *****)
       Init := false;

      IF data_Ini THEN                            (* Параметрам требуется переинициализация. *)
          strAI.dLL                := dLL;
          strAI.dHL                := dHL;
          strAI.dLA                := dLA;
          strAI.dHA                := dHA;
          strAI.dLW                := dLW;
          strAI.dHW                := dHW;
          strAI.ISVALIDREF_LA      := ISVALIDREF_LA;
          strAI.ISVALIDREF_HA      := ISVALIDREF_HA;
          strAI.ISVALIDREF_LW      := ISVALIDREF_LW;
          strAI.ISVALIDREF_HW      := ISVALIDREF_HW;
          strAI.delayLA            := delayLA;
          strAI.delayLW            := delayLW;
          strAI.delayHW            := delayHW;
          strAI.delayHA            := delayHA;
          strAI.inpLL              := inpLL;
          strAI.inpHL              := inpHL;
          strAI.CurrentShotCircuit := CurrentShotCircuit;
          strAI.CurrentBreakCircuit:= CurrentBreakCircuit;
          strAI.dMaxChangeSpeed     := dMaxChangeSpeed;
          strAI.dMaxChangeSpeedDown := dMaxChangeSpeedDown;
          strAI.histeresis         := histeresis;
          strAI.aperturFilter      := aperturFilter;
          strAI.exponentialFilter  := exponentialFilter;
          strAI.rassoglasovanie    := rassoglasovanie;
          strAI.rassoglasovanie    := rassoglasovanie;

          data_Ini:=false;
          Init := TRUE;
       END_IF;
    IF Init THEN
          dLL:= 0.0;
          dHL:= 0.0;
          dLA:= 0.0;
          dHA:= 0.0;
          dLW:= 0.0;
          dHW:= 0.0;
          inpLL:= 4000.0;
          inpHL:= 20000.0;
          CurrentShotCircuit:= 21000.0;
          CurrentBreakCircuit:= 3700.0;
          ISVALIDREF_LA:= false;
          ISVALIDREF_HA:= false;
          ISVALIDREF_LW:= false;
          ISVALIDREF_HW:= false;
          delayLA:= T#0S;
          delayLW:= T#0S;
          delayHW:= T#0S;
          delayHA:= T#0S;
          dMaxChangeSpeed:= 0.0;
          dMaxChangeSpeedDown:= 0.0;
          histeresis:= 0.0;
          aperturFilter:= 0.0;
          exponentialFilter:= 0.0;
          rassoglasovanie:= 0.0;
        END_IF;
END_FUNCTION_BLOCK

FUNCTION EnableAiLimits : BOOL
  VAR_IN_OUT
    ai : AiConfig;
  END_VAR

  ai.Pmasla_posle_GNS.Disabled_LA:=FALSE;
   ai.Pmasla_posle_GNS.Disabled_LW:=FALSE;
   ai.Pmasla_posle_NU.Disabled_LW:=FALSE;
   ai.Tmasla_MB.Disabled_LA:=FALSE;
   ai.Tmasla_MB.Disabled_LW:=FALSE;
END_FUNCTION

FUNCTION DisableAiLimits : BOOL
  VAR_IN_OUT
    ai : AiConfig;
  END_VAR

  ai.Pmasla_posle_GNS.Disabled_LA:=TRUE;
   ai.Pmasla_posle_GNS.Disabled_LW:=TRUE;
   ai.Pmasla_posle_NU.Disabled_LW:=TRUE;
   ai.Tmasla_MB.Disabled_LA:=TRUE;
   ai.Tmasla_MB.Disabled_LW:=TRUE;
END_FUNCTION

FUNCTION_BLOCK TestProtectionAlg
  VAR_IN_OUT
    StrAlg : struct_Alg;
  END_VAR
  VAR
    _sunpackerCommand : fb_sunpackerCommand;
    source : BYTE;
    cmd : BYTE;
    lastCmd : BYTE;
    source_for_Status : BYTE;
    cmd_for_Status : BYTE;
    command_error_for_Status : BYTE;
    resetCmdTimer : TON;
    resetCmdTimerPriznak : BOOL;
  END_VAR
  VAR_EXTERNAL
    ai : AiConfig;
    protectManager : struct_ProtectionsManager;
    algManager : struct_AlgoritmsManager;
    ModeGpa : TYPE_ModeGpa;
    PMcommand : TYPE_CommandsPotectionsManager;
    IM : ImConfig;
  END_VAR

  StrAlg.CanRun := StrAlg.inCanRun;
  StrAlg.OpcCommandsDisabled := StrAlg.inOpcCommandsDisabled;

  (* ---- Если управление с ВУ заблокировано, то передаем команду из алгоритма ---- *)
  IF StrAlg.inOpcCommandsDisabled THEN
  	StrAlg.inCommand := StrAlg.inCommand_Alg;
  ELSE (* иначе передаем команду с АРМа*)
  	StrAlg.inCommand := StrAlg.inCommand_ARM;
  END_IF;

  _sunpackerCommand(command := StrAlg.inCommand);
  	source := _sunpackerCommand.source;
  	cmd := _sunpackerCommand.cmd;

  IF cmd <> 0 AND lastCmd <> cmd AND (((NOT StrAlg.opcCommandsDisabled) AND source > 0) OR source = 0) then
  	CASE BYTE_TO_INT(cmd) OF
  		(*cmdRun*) 1: 	IF (StrAlg.CanRun) THEN
  					StrAlg.isRuning := TRUE;
  					StrAlg.isEnded := FALSE;
  					StrAlg.hasError 	:= FALSE;
                                               (*****************       OnRun       *****************)
                                                        algManager.nMode:=ModeGpa.MODE_TESTAZ;
                                                        protectManager.inCommand:=PMcommand.CheckProtections;
  					    EnableAiLimits(ai);
                                                        (*IM.SingleSignals.P_oil_low.Disabled_Sig:=FALSE;*)
                                                        (*IM.SingleSignals.dP_oilgaz_low.Disabled_Sig:=FALSE;*)
                                                    (*StrAlg.inOpcCommandsDisabled:=FALSE;*)
  					cmd_for_Status := cmd;
  					source_for_Status := source;
  					command_error_for_Status := 0;
  				ELSE
  					StrAlg.isRuning := FALSE;
  					StrAlg.isEnded := FALSE;
  					StrAlg.hasError 	:= FALSE;

  					cmd_for_Status := 0;
  					source_for_Status := source;
  					command_error_for_Status := cmd;
  				END_IF;
  		(*cmdReset*) 2: 	StrAlg.isRuning := FALSE;
  				StrAlg.isEnded := FALSE;
  				StrAlg.hasError 	:= FALSE;
                                          (*****************       OnReset       *****************)
                                                    DisableAiLimits(ai);
                                                    (*IM.SingleSignals.P_oil_low.Disabled_Sig:=TRUE;
                                                    IM.SingleSignals.dP_oilgaz_low.Disabled_Sig:=TRUE;*)
                                                    protectManager.inCommand:=PMcommand.RestartAllProtections;
                                                    algManager.nMode:=ModeGpa.MODE_STOP;

  				cmd_for_Status := cmd;
  				source_for_Status := source;
  				command_error_for_Status := 0;
  	END_CASE;
  	resetCmdTimer(IN := false);
  	resetCmdTimerPriznak := TRUE;
  END_IF;
  lastCmd := cmd;

  resetCmdTimer(IN := resetCmdTimerPriznak, PT := T#5S);
  IF resetCmdTimer.Q THEN
  	resetCmdTimerPriznak := FALSE;
  	source_for_Status := 0;
  	cmd_for_Status := 0;
  	command_error_for_Status := 0;
  END_IF;

  StrAlg.status :=  SHL(BYTE_TO_DWORD(source_for_Status), 29)
  			OR SHL(BYTE_TO_DWORD(cmd_for_Status), 26)
  			OR SHL(BYTE_TO_DWORD(command_error_for_Status), 23)
  			OR SHL(BOOL_TO_DWORD(StrAlg.OpcCommandsDisabled ), 21)
  			OR SHL(BOOL_TO_DWORD(StrAlg.hasError),4)
  			OR SHL(BOOL_TO_DWORD(StrAlg.CanRun),2)
  			OR SHL(BOOL_TO_DWORD(StrAlg.isEnded),1)
  			OR BOOL_TO_DWORD(StrAlg.isRuning);
END_FUNCTION_BLOCK

FUNCTION_BLOCK TestImAlg
  VAR_IN_OUT
    StrAlg : struct_Alg;
  END_VAR
  VAR
    _sunpackerCommand : fb_sunpackerCommand;
    source : BYTE;
    cmd : BYTE;
    lastCmd : BYTE;
    source_for_Status : BYTE;
    cmd_for_Status : BYTE;
    command_error_for_Status : BYTE;
    resetCmdTimer : TON;
    resetCmdTimerPriznak : BOOL;
  END_VAR
  VAR_EXTERNAL
    protectManager : struct_ProtectionsManager;
    algManager : struct_AlgoritmsManager;
    ModeGpa : TYPE_ModeGpa;
    PMcommand : TYPE_CommandsPotectionsManager;
    IM : ImConfig;
  END_VAR

  StrAlg.CanRun := StrAlg.inCanRun;
  StrAlg.OpcCommandsDisabled := StrAlg.inOpcCommandsDisabled;

  (* ---- Если управление с ВУ заблокировано, то передаем команду из алгоритма ---- *)
  IF StrAlg.inOpcCommandsDisabled THEN
  	StrAlg.inCommand := StrAlg.inCommand_Alg;
  ELSE (* иначе передаем команду с АРМа*)
  	StrAlg.inCommand := StrAlg.inCommand_ARM;
  END_IF;

  _sunpackerCommand(command := StrAlg.inCommand);
  	source := _sunpackerCommand.source;
  	cmd := _sunpackerCommand.cmd;

  IF cmd <> 0 AND lastCmd <> cmd AND (((NOT StrAlg.opcCommandsDisabled) AND source > 0) OR source = 0) then
  	CASE BYTE_TO_INT(cmd) OF
  		(*cmdRun*) 1: 	IF (StrAlg.CanRun) THEN
  					StrAlg.isRuning := TRUE;
  					StrAlg.isEnded := FALSE;
  					StrAlg.hasError 	:= FALSE;
                                               (*****************       OnRun       *****************)

                                                        algManager.nMode:=ModeGpa.MODE_TESTIM;
  					    UnBlockAllIM(IM);

                                                    (*StrAlg.inOpcCommandsDisabled:=FALSE;*)
  					cmd_for_Status := cmd;
  					source_for_Status := source;
  					command_error_for_Status := 0;
  				ELSE
  					StrAlg.isRuning := FALSE;
  					StrAlg.isEnded := FALSE;
  					StrAlg.hasError 	:= FALSE;

  					cmd_for_Status := 0;
  					source_for_Status := source;
  					command_error_for_Status := cmd;
  				END_IF;
  		(*cmdReset*) 2: 	StrAlg.isRuning := FALSE;
  				StrAlg.isEnded := FALSE;
  				StrAlg.hasError 	:= FALSE;
                                          (*****************       OnReset       *****************)
                                                    BlockAllIM(IM);
                                                    algManager.nMode:=ModeGpa.MODE_STOP;

  				cmd_for_Status := cmd;
  				source_for_Status := source;
  				command_error_for_Status := 0;
  	END_CASE;
  	resetCmdTimer(IN := false);
  	resetCmdTimerPriznak := TRUE;
  END_IF;
  lastCmd := cmd;

  resetCmdTimer(IN := resetCmdTimerPriznak, PT := T#5S);
  IF resetCmdTimer.Q THEN
  	resetCmdTimerPriznak := FALSE;
  	source_for_Status := 0;
  	cmd_for_Status := 0;
  	command_error_for_Status := 0;
  END_IF;

  StrAlg.status :=  SHL(BYTE_TO_DWORD(source_for_Status), 29)
  			OR SHL(BYTE_TO_DWORD(cmd_for_Status), 26)
  			OR SHL(BYTE_TO_DWORD(command_error_for_Status), 23)
  			OR SHL(BOOL_TO_DWORD(StrAlg.OpcCommandsDisabled ), 21)
  			OR SHL(BOOL_TO_DWORD(StrAlg.hasError),4)
  			OR SHL(BOOL_TO_DWORD(StrAlg.CanRun),2)
  			OR SHL(BOOL_TO_DWORD(StrAlg.isEnded),1)
  			OR BOOL_TO_DWORD(StrAlg.isRuning);
END_FUNCTION_BLOCK

FUNCTION_BLOCK fb_AutoTenAlg
  VAR_IN_OUT
    StrAlg : struct_Alg;
    PNS : struct_Switch;
    TEN : struct_Switch;
  END_VAR
  VAR_INPUT
    T_masla : struct_AI;
    Uroven_masla : struct_AI;
    offTemperature : struct_AnalogParametr;
  END_VAR
  VAR
    _sunpackerCommand : fb_sunpackerCommand;
    _statusAi : TYPE_StatusAi;
    _statusDualInput : TYPE_statusDualInput;
    _commandDualInput : TYPE_commandDualInput;
    source : BYTE;
    cmd : BYTE;
    lastCmd : BYTE;
    source_for_Status : BYTE;
    cmd_for_Status : BYTE;
    command_error_for_Status : BYTE;
    resetCmdTimer : TON;
    resetCmdTimerPriznak : BOOL;
    onInit : BOOL;
  END_VAR

  IF NOT onInit THEN
  StrAlg.inCanRun:=TRUE;
  onInit:=TRUE;
  END_IF;

  IF StrAlg.isRuning THEN

  IF ((T_masla.interval >= _statusAi.normal) AND (T_masla.value > offTemperature.Value)) OR
  ((Uroven_masla.interval >= _statusAi.normal) AND (Uroven_masla.value < Uroven_masla.LA)) OR
  (PNS.onStatus=_statusDualInput.STATUS_OFF) THEN

        TEN.inOpcCommandsDisabled:=TRUE;

  	IF TEN.onStatus = _statusDualInput.STATUS_ON THEN
            TEN.inCommand_Alg:=BYTE_TO_WORD(_commandDualInput.CMD_OFF);
  	END_IF;

  ELSIF PNS.onStatus = _statusDualInput.STATUS_ON THEN
        TEN.inOpcCommandsDisabled:=FALSE;
  END_IF;

  END_IF;

  StrAlg.CanRun := StrAlg.inCanRun;
  StrAlg.hasError := TEN.CommandFault OR (T_masla.interval < _statusAi.normal) OR (Uroven_masla.interval < _statusAi.normal);

  StrAlg.OpcCommandsDisabled := StrAlg.inOpcCommandsDisabled;

  (* ---- Если управление с ВУ заблокировано, то  передаем команду из алгоритма ---- *)
  IF StrAlg.inOpcCommandsDisabled THEN
  	StrAlg.inCommand := StrAlg.inCommand_Alg;
  ELSE (* иначе передаем команду с АРМа*)
  	StrAlg.inCommand := StrAlg.inCommand_ARM;
  END_IF;

  _sunpackerCommand(command := StrAlg.inCommand);
  	source := _sunpackerCommand.source;
  	cmd := _sunpackerCommand.cmd;

  IF cmd <> 0 AND lastCmd <> cmd AND (((NOT StrAlg.opcCommandsDisabled) AND source > 0) OR source = 0) then
  	CASE BYTE_TO_INT(cmd) OF
  		(*cmdRun*) 1: 	IF StrAlg.CanRun AND NOT StrAlg.hasError THEN
  					StrAlg.isRuning := TRUE;
  					StrAlg.isEnded := FALSE;
  					(*StrAlg.hasError := FALSE;*)

                                                    (*****************       OnRun       *****************)
                                                    IF StrAlg.inOpcCommandsDisabled THEN
  		                              StrAlg.inOpcCommandsDisabled:=FALSE;
                                                    END_IF;
  					cmd_for_Status := cmd;
  					source_for_Status := source;
  					command_error_for_Status := 0;
  				ELSE
  					StrAlg.isRuning := FALSE;
  					StrAlg.isEnded := FALSE;
  					(*StrAlg.hasError 	:= FALSE;*)

  					cmd_for_Status := 0;
  					source_for_Status := source;
  					command_error_for_Status := cmd;
  				END_IF;
  		(*cmdReset*) 2: 	StrAlg.isRuning := FALSE;
  				StrAlg.isEnded := FALSE;
  				(*StrAlg.hasError 	:= FALSE;*)

                                          (*****************       OnReset       *****************)
                                          TEN.inOpcCommandsDisabled:=TRUE;
                                          TEN.inCommand_Alg:=BYTE_TO_WORD(_commandDualInput.CMD_OFF);

  				cmd_for_Status := cmd;
  				source_for_Status := source;
  				command_error_for_Status := 0;
  	END_CASE;
  	resetCmdTimer(IN := false);
  	resetCmdTimerPriznak := TRUE;
  END_IF;
  lastCmd := cmd;

  resetCmdTimer(IN := resetCmdTimerPriznak, PT := T#5S);
  IF resetCmdTimer.Q THEN
  	resetCmdTimerPriznak := FALSE;
  	source_for_Status := 0;
  	cmd_for_Status := 0;
  	command_error_for_Status := 0;
  END_IF;

  (*TODO: TYPE PROGRAM CODE HERE*)
  StrAlg.status :=  SHL(BYTE_TO_DWORD(source_for_Status), 29)
  			OR SHL(BYTE_TO_DWORD(cmd_for_Status), 26)
  			OR SHL(BYTE_TO_DWORD(command_error_for_Status), 23)
  			OR SHL(BOOL_TO_DWORD(StrAlg.OpcCommandsDisabled ), 21)
  			OR SHL(BOOL_TO_DWORD(StrAlg.hasError),4)
  			OR SHL(BOOL_TO_DWORD(StrAlg.CanRun),2)
  			OR SHL(BOOL_TO_DWORD(StrAlg.isEnded),1)
  			OR BOOL_TO_DWORD(StrAlg.isRuning);
END_FUNCTION_BLOCK

FUNCTION_BLOCK fb_AutoPnsAlg
  VAR_IN_OUT
    StrAlg : struct_Alg;
    Nasos : struct_Switch;
  END_VAR
  VAR_INPUT
    diPlow : struct_singleSignal;
    Poil : struct_AI;
    Ust_Run : struct_AnalogParametr;
    Ust_Stop : struct_AnalogParametr;
  END_VAR
  VAR
    _sunpackerCommand : fb_sunpackerCommand;
    _statusAi : TYPE_StatusAi;
    _statusDualInput : TYPE_statusDualInput;
    _commandDualInput : TYPE_commandDualInput;
    source : BYTE;
    cmd : BYTE;
    lastCmd : BYTE;
    source_for_Status : BYTE;
    cmd_for_Status : BYTE;
    command_error_for_Status : BYTE;
    resetCmdTimer : TON;
    resetCmdTimerPriznak : BOOL;
    onInit : BOOL;
    onTrig : R_TRIG;
    offTrig : R_TRIG;
    waitOn : TON;
    waitOff : TON;
  END_VAR
  VAR_EXTERNAL
    AlgTimers : struct_AlgTimers;
  END_VAR

  IF NOT onInit THEN
  StrAlg.inOpcCommandsDisabled:=TRUE;
  StrAlg.inCanRun:=TRUE;
  onInit:=TRUE;
  END_IF;

  IF StrAlg.isRuning THEN

  StrAlg.hasError := Nasos.CommandFault OR (Poil.interval < _statusAi.normal OR NOT diPlow.reliability);

      IF (Poil.Interval >= _statusAi.normal) THEN
      waitOn(IN:=Poil.Value <= Ust_Run.value OR diPlow.q, PT := T#1S);
      waitOff(IN:= Poil.Value >= Ust_Stop.value, PT := T#300S);

      ELSE
      waitOn(IN:=diPlow.Q, PT := T#1S);
      END_IF;

  onTrig(CLK:=waitOn.Q);
  offTrig(CLK:=waitOff.Q);
      IF (Poil.Value>=Ust_Stop.value) AND Nasos.inopcCommandsDisabled THEN
          Nasos.inopcCommandsDisabled:=FALSE;
      END_IF;

      IF onTrig.Q THEN
      Nasos.inopcCommandsDisabled:=TRUE;
      Nasos.inCommand_Alg:=BYTE_TO_WORD(_commandDualInput.CMD_ON);
      END_IF;

      IF offTrig.Q THEN
          IF NOT (Nasos.onStatus=_statusDualInput.STATUS_OFF) THEN
          Nasos.inopcCommandsDisabled:=TRUE;
          Nasos.inCommand_Alg:=BYTE_TO_WORD(_commandDualInput.CMD_OFF);
          END_IF;
      END_IF;

  AlgTimers.AutoPns_OnTimer:=UDINT_TO_UINT(TIME_TO_UDINT(waitOn.PT - waitOn.ET)/1000);
  AlgTimers.AutoPns_OffTimer:=UDINT_TO_UINT(TIME_TO_UDINT(waitOff.PT -waitOff.ET)/1000);

  END_IF;

  StrAlg.CanRun := StrAlg.inCanRun;

  StrAlg.OpcCommandsDisabled := StrAlg.inOpcCommandsDisabled;

  (* ---- Если управление с ВУ заблокировано, то  передаем команду из алгоритма ---- *)
  IF StrAlg.inOpcCommandsDisabled THEN
  	StrAlg.inCommand := StrAlg.inCommand_Alg;
  ELSE (* иначе передаем команду с АРМа*)
  	StrAlg.inCommand := StrAlg.inCommand_ARM;
  END_IF;

  _sunpackerCommand(command := StrAlg.inCommand);
  	source := _sunpackerCommand.source;
  	cmd := _sunpackerCommand.cmd;

  IF cmd <> 0 AND lastCmd <> cmd AND (((NOT StrAlg.opcCommandsDisabled) AND source > 0) OR source = 0) then
  	CASE BYTE_TO_INT(cmd) OF
  		(*cmdRun*) 1: 	IF (StrAlg.CanRun) THEN
  					StrAlg.isRuning := TRUE;
  					StrAlg.isEnded := FALSE;
  					StrAlg.hasError := FALSE;
  					(*****************       OnRun       *****************)

  					cmd_for_Status := cmd;
  					source_for_Status := source;
  					command_error_for_Status := 0;
  				ELSE
  					StrAlg.isRuning := FALSE;
  					StrAlg.isEnded := FALSE;
  					StrAlg.hasError 	:= FALSE;

  					cmd_for_Status := 0;
  					source_for_Status := source;
  					command_error_for_Status := cmd;
  				END_IF;
  		(*cmdReset*) 2: 	StrAlg.isRuning := FALSE;
  				StrAlg.isEnded := FALSE;
  				StrAlg.hasError 	:= FALSE;

                                           (*****************       OnReset       *****************)
                                          waitOn(in:=FALSE);
                                          waitOff(in:=FALSE);
                                          AlgTimers.AutoPns_OffTimer:=UDINT_TO_UINT(TIME_TO_UDINT(waitOff.pt -waitOff.ET)/1000);

  				cmd_for_Status := cmd;
  				source_for_Status := source;
  				command_error_for_Status := 0;
  	END_CASE;
  	resetCmdTimer(IN := false);
  	resetCmdTimerPriznak := TRUE;
  END_IF;
  lastCmd := cmd;

  resetCmdTimer(IN := resetCmdTimerPriznak, PT := T#5S);
  IF resetCmdTimer.Q THEN
  	resetCmdTimerPriznak := FALSE;
  	source_for_Status := 0;
  	cmd_for_Status := 0;
  	command_error_for_Status := 0;
  END_IF;

  (*TODO: TYPE PROGRAM CODE HERE*)
  StrAlg.status :=  SHL(BYTE_TO_DWORD(source_for_Status), 29)
  			OR SHL(BYTE_TO_DWORD(cmd_for_Status), 26)
  			OR SHL(BYTE_TO_DWORD(command_error_for_Status), 23)
  			OR SHL(BOOL_TO_DWORD(StrAlg.OpcCommandsDisabled ), 21)
  			OR SHL(BOOL_TO_DWORD(StrAlg.hasError),4)
  			OR SHL(BOOL_TO_DWORD(StrAlg.CanRun),2)
  			OR SHL(BOOL_TO_DWORD(StrAlg.isEnded),1)
  			OR BOOL_TO_DWORD(StrAlg.isRuning);
END_FUNCTION_BLOCK

FUNCTION_BLOCK fb_AutoAvomAlg
  VAR_IN_OUT
    StrAlg : struct_Alg;
    im1 : struct_Switch;
    im2 : struct_Switch;
  END_VAR
  VAR_INPUT
    ai : struct_AI;
  END_VAR
  VAR_IN_OUT
    on1Temperature : struct_AnalogParametr;
    on2Temperature : struct_AnalogParametr;
    hystereses : struct_AnalogParametr;
  END_VAR
  VAR
    _sunpackerCommand : fb_sunpackerCommand;
    _statusAi : TYPE_StatusAi;
    _statusDualInput : TYPE_statusDualInput;
    _commandDualInput : TYPE_commandDualInput;
    source : BYTE;
    cmd : BYTE;
    lastCmd : BYTE;
    source_for_Status : BYTE;
    cmd_for_Status : BYTE;
    command_error_for_Status : BYTE;
    resetCmdTimer : TON;
    resetCmdTimerPriznak : BOOL;
    onInit : BOOL;
  END_VAR

  (*
  IF NOT onInit THEN
  StrAlg.inCanRun:=TRUE;
  onInit:=TRUE;
  END_IF;
  *)

  IF StrAlg.isRuning THEN

  StrAlg.hasError := im1.CommandFault OR im2.CommandFault OR (ai.interval<_statusAi.normal);

      IF (ai.interval>=_statusAi.normal) THEN

            IF (ai.value>= on1Temperature.Value) THEN
                IF im1.onStatus <> _statusDualInput.STATUS_ON THEN
  	       im1.inCommand_Alg:=BYTE_TO_WORD(_commandDualInput.CMD_ON); (*cmd_on*)
                END_IF;
            END_IF;

            IF  ai.value < (on1Temperature.Value - hystereses.Value) THEN
                IF im1.onStatus <> _statusDualInput.STATUS_OFF THEN
  	       im1.inCommand_Alg:=BYTE_TO_WORD(_commandDualInput.CMD_OFF);
                END_IF;
            END_IF;

             IF (ai.value>= on2Temperature.Value) THEN
                IF im2.onStatus <> _statusDualInput.STATUS_ON THEN
  	       im2.inCommand_Alg:=BYTE_TO_WORD(_commandDualInput.CMD_ON); (*cmd_on*)
                END_IF;
            END_IF;

            IF  ai.value < (on2Temperature.Value - hystereses.Value) THEN
                IF im2.onStatus <> _statusDualInput.STATUS_OFF THEN
  	       im2.inCommand_Alg:=BYTE_TO_WORD(_commandDualInput.CMD_OFF);
                END_IF;
            END_IF;
       END_IF;

  END_IF;

  StrAlg.CanRun := StrAlg.inCanRun;

  StrAlg.OpcCommandsDisabled := StrAlg.inOpcCommandsDisabled;

  (* ---- Если управление с ВУ заблокировано, то  передаем команду из алгоритма ---- *)
  IF StrAlg.inOpcCommandsDisabled THEN
  	StrAlg.inCommand := StrAlg.inCommand_Alg;
  ELSE (* иначе передаем команду с АРМа*)
  	StrAlg.inCommand := StrAlg.inCommand_ARM;
  END_IF;

  _sunpackerCommand(command := StrAlg.inCommand);
  	source := _sunpackerCommand.source;
  	cmd := _sunpackerCommand.cmd;

  IF cmd <> 0 AND lastCmd <> cmd AND (((NOT StrAlg.opcCommandsDisabled) AND source > 0) OR source = 0) then
  	CASE BYTE_TO_INT(cmd) OF
  		(*cmdRun*) 1: 	IF (StrAlg.CanRun) THEN
  					StrAlg.isRuning := TRUE;
  					StrAlg.isEnded := FALSE;
  					StrAlg.hasError := FALSE;
                                                    StrAlg.inOpcCommandsDisabled:=FALSE;
  					im1.inOpcCommandsDisabled:=TRUE;
                                                    im2.inOpcCommandsDisabled:=TRUE;
  					cmd_for_Status := cmd;
  					source_for_Status := source;
  					command_error_for_Status := 0;
  				ELSE
  					StrAlg.isRuning := FALSE;
  					StrAlg.isEnded := FALSE;
  					StrAlg.hasError 	:= FALSE;

  					cmd_for_Status := 0;
  					source_for_Status := source;
  					command_error_for_Status := cmd;
  				END_IF;
  		(*cmdReset*) 2: 	StrAlg.isRuning := FALSE;
  				StrAlg.isEnded := FALSE;
  				StrAlg.hasError 	:= FALSE;
                                          StrAlg.inOpcCommandsDisabled:=FALSE;
                                          im1.inOpcCommandsDisabled:=FALSE;
                                          im2.inOpcCommandsDisabled:=FALSE;
                                          im1.inCommand_Alg:=0;
                                          im2.inCommand_Alg:=0;
  				cmd_for_Status := cmd;
  				source_for_Status := source;
  				command_error_for_Status := 0;
  	END_CASE;
  	resetCmdTimer(IN := false);
  	resetCmdTimerPriznak := TRUE;
  END_IF;
  lastCmd := cmd;

  resetCmdTimer(IN := resetCmdTimerPriznak, PT := T#5S);
  IF resetCmdTimer.Q THEN
  	resetCmdTimerPriznak := FALSE;
  	source_for_Status := 0;
  	cmd_for_Status := 0;
  	command_error_for_Status := 0;
  END_IF;

  (*TODO: TYPE PROGRAM CODE HERE*)
  StrAlg.status :=  SHL(BYTE_TO_DWORD(source_for_Status), 29)
  			OR SHL(BYTE_TO_DWORD(cmd_for_Status), 26)
  			OR SHL(BYTE_TO_DWORD(command_error_for_Status), 23)
  			OR SHL(BOOL_TO_DWORD(StrAlg.OpcCommandsDisabled ), 21)
  			OR SHL(BOOL_TO_DWORD(StrAlg.hasError),4)
  			OR SHL(BOOL_TO_DWORD(StrAlg.CanRun),2)
  			OR SHL(BOOL_TO_DWORD(StrAlg.isEnded),1)
  			OR BOOL_TO_DWORD(StrAlg.isRuning);
END_FUNCTION_BLOCK
